// TIA Portal project "T2" (V17)

(* hardware
DEVICE "S7-1500/ET200MP station_1"  S7-1500 station
   slot 0: "Rail_0"  Rack  6ES7 590-1***0-0AA0
   slot 1: "PLC_1"  CPU 1511-1 PN  6ES7 511-1AK01-0AB0  V2.9
      slot 3: "CPU display_1"  6ES7591-1AA00-0AA0
      slot 32768: "PROFINET interface_1"  X1
         slot 32769: "Port_1"  X1 P1
         slot 32770: "Port_2"  X1 P2
      slot 34817: "Virtual CP interface port_1"  Virtual CP interface port  Virtual CP interface port
   slot 2: "DI 32x24VDC SNK/SRC / DQ 32x24VDC/0.3A SNK BA_1"  DI 32x24VDC SNK/SRC / DQ 32x24VDC/0.3A SNK BA  6ES7 523-1BP50-0AA0  V1.0
DEVICE "HMI_1"  TP1500 Comfort PRO
   slot 0: "HMI_1"  TP1500 Comfort PRO  6AV2 124-0QC24-1AXx  17.0.0.0
   slot 1: "HMI_RT_2"  TP1500 Comfort PRO  6AV2 124-0QC24-1AXx  17.0.0.0
   slot 5: "HMI_1.IE_CP_1"  PROFINET Interface  17.0.0.0
      slot 1: "PROFINET Interface_1"  PROFINET Interface
         slot 1: "Port_1"  Port
         slot 2: "Port_2"  Port
   slot 6: "HMI_1.IE_CP_2"  PROFINET Interface  17.0.0.0
      slot 1: "PROFINET Interface_GBit"  PROFINET Interface
         slot 1: "Port_1"  Port
   slot 7: "HMI_1.MPI/DP_CP_1"  MPI/DP Interface  17.0.0.0
*)

// ===== PLC "PLC_1"  CPU 1511-1 PN =====

VAR_GLOBAL   // PLC tag table "Default tag table"
   "System_Byte" AT %MB500 : Byte;
   "FirstScan" AT %M500.0 : Bool;
   "DiagStatusUpdate" AT %M500.1 : Bool;
   "AlwaysTRUE" AT %M500.2 : Bool;
   "AlwaysFALSE" AT %M500.3 : Bool;
   "OPC_Marcha" AT %I0.0 : Bool;
   "OPC_Paro" AT %I0.1 : Bool;
   "Mantenimineto_Fin" AT %M0.0 : Bool;
   "Act_Mantenimiento" AT %M0.1 : Bool;
   "Proceso_Activo" AT %M0.2 : Bool;
   "OPC_SPress_VAC" AT %I0.2 : Bool;
   "OPC_S1_VAC" AT %I0.3 : Bool;
   "OPC_S3_VAC" AT %I0.4 : Bool;
   "OPC_S4_VAC" AT %I0.5 : Bool;
   "OPC_S5_VAC" AT %I0.6 : Bool;
   "OPC_S_VAC_A_Buena" AT %I0.7 : Bool;
   "OPC_S_VAC_A_Mala" AT %I1.0 : Bool;
   "OPC_S_VAC_B" AT %I1.1 : Bool;
   "P_REC_MAQ_CAL_VAC" AT %M0.6 : Bool;
   "P_REC_MAQ_CAL_SOP" AT %M0.7 : Bool;
   "P_REC_MAQ_CAL_EMB" AT %M1.0 : Bool;
   "OPC_Emisor_Vacunas" AT %Q0.0 : Bool;
   "OPC_QC2_VAC" AT %Q0.2 : Bool;
   "OPC_QC3_VAC" AT %Q0.3 : Bool;
   "Pieza_Enviada_MAQ_5_VAC" AT %M3.0 : Bool;
   "VACUNA_ESPERANDO_SOPORTE" AT %M3.2 : Bool;
   "Vacuna_en_Soporte" AT %M3.3 : Bool;
   "Pieza_Enviada_MAQ_5_SOP" AT %M4.1 : Bool;
   "SOPORTE_ESPERANDO_VACUNA" AT %M4.2 : Bool;
   "ACT_EMP_1" AT %M4.6 : Bool;
   "P_Enviada_EMP1" AT %M4.7 : Bool;
   "ACT_EMP_2" AT %M5.0 : Bool;
   "P_Enviada_EMP2" AT %M5.1 : Bool;
   "Transfer_EMP_VACSOP1_Libre" AT %M5.2 : Bool;
   "Transfer_EMP_VACSOP2_Libre" AT %M5.4 : Bool;
   "Vacuna_A" AT %M6.0 : Bool;
   "Vacuna_B" AT %M6.1 : Bool;
   "Soporte_A" AT %M6.2 : Bool;
   "Soporte_B" AT %M6.3 : Bool;
   "Embalaje_A" AT %M6.4 : Bool;
   "Embalaje_B" AT %M6.5 : Bool;
   "Pieza_Enviada_MAQ_5_EMB" AT %M7.2 : Bool;
   "P_Enviada_EMB_EMB" AT %M7.3 : Bool;
   "Cinta_7_EMB_Libre" AT %M7.4 : Bool;
   "Activar_TRansfer_3_EMP" AT %M7.5 : Bool;
   "Act_Cinta_7_EMP" AT %M7.6 : Bool;
   "Transfer_3_EMP_Libre" AT %M7.7 : Bool;
   "Transfer_2_EMP_EMBSOPVAC_Libre" AT %M8.0 : Bool;
   "Trasnfer_2_EMPSOPVAC_Libre" AT %M8.2 : Bool;
   "Trasnfer_1_EMPSOPVAC_Libre" AT %M8.3 : Bool;
   "Act_Maq_1_EMBSOPVAC" AT %M8.4 : Bool;
   "Act_Maq_2_EMBSOPVAC" AT %M8.5 : Bool;
   "EMP1_EMBSOPVAC_Libre" AT %M8.6 : Bool;
   "Esperando_Embalaje" AT %M8.7 : Bool;
   "Vacuna_Lista" AT %M9.4 : Bool;
   "Empaquetar_vacuna" AT %M9.5 : Bool;
   "Empaquetar_Soporte" AT %M9.6 : Bool;
   "Vacuna_Empaquetada" AT %M9.7 : Bool;
   "Soporte_Empaquetado" AT %M10.0 : Bool;
   "Soporte_Listo" AT %M10.1 : Bool;
   "OPC_SETA" AT %I1.2 : Bool;
   "Act_Mantenimiento_Emergencia" AT %M10.2 : Bool;
   "Act_Vaciado" AT %M10.3 : Bool;
   "Emergencia" AT %M10.4 : Bool;
   "Fin_Vaciado" AT %M10.5 : Bool;
   "OPC_Reset" AT %I1.3 : Bool;
   "OPC_Resume" AT %I2.3 : Bool;
   "HMI_Marcha" AT %M10.6 : Bool;
   "ContadorPiezasFinalizadas" AT %MW12 : Int;
   "OPC_QC4_VAC" AT %Q0.4 : Bool;
   "OPC_QC5_VAC" AT %Q0.5 : Bool;
   "OPC_QC6_VAC" AT %Q0.6 : Bool;
   "OPC_QC7_VAC" AT %Q0.7 : Bool;
   "OPC_QTRANS1_VAC" AT %Q1.0 : Bool;
   "OPC_QTRANS2_VAC" AT %Q1.1 : Bool;
   "OPC_QHOR_VAC" AT %Q1.2 : Bool;
   "OPC_QBAJ_VAC" AT %Q1.3 : Bool;
   "OPC_QGRIP_VAC" AT %Q1.4 : Bool;
   "OPC_CLAMP1_VAC" AT %Q1.5 : Bool;
   "HaySoporte" AT %M3.1 : Bool;
   "HayVacuna" AT %M3.4 : Bool;
   "VacunaEnSoporte" AT %M3.5 : Bool;
   "OPC_SPress_SOP" AT %I1.4 : Bool;
   "OPC_S1_SOP" AT %I1.5 : Bool;
   "OPC_S3_SOP" AT %I1.6 : Bool;
   "OPC_S4_SOP" AT %I1.7 : Bool;
   "OPC_S5_SOP" AT %I2.0 : Bool;
   "OPC_S_SOP_A_Buena" AT %I2.1 : Bool;
   "OPC_S_SOP_A_Mala" AT %I2.2 : Bool;
   "OPC_S_SOP_B" AT %I2.4 : Bool;
   "OPC_Emisor_SOP" AT %Q1.7 : Bool;
   "OPC_QC1_SOP" AT %Q2.0 : Bool;
   "OPC_QC2_SOP" AT %Q2.1 : Bool;
   "OPC_QC3_SOP" AT %Q2.2 : Bool;
   "OPC_QC4_SOP" AT %Q2.3 : Bool;
   "OPC_QC5_SOP" AT %Q2.4 : Bool;
   "OPC_QC6_SOP" AT %Q2.5 : Bool;
   "OPC_QC7_SOP" AT %Q2.6 : Bool;
   "OPC_QTRANS1_SOP" AT %Q2.7 : Bool;
   "OPC_QTRANS2_SOP" AT %Q3.0 : Bool;
   "OPC_QHOR_SOP" AT %Q3.1 : Bool;
   "OPC_QBAJ_SOP" AT %Q3.2 : Bool;
   "OPC_QGRIP_SOP" AT %Q3.3 : Bool;
   "OPC_CLAMP1_SOP" AT %Q3.4 : Bool;
   "OPC_SUBCLAMP1_SOP" AT %Q3.5 : Bool;
   "OPC_QC8_SOP" AT %Q3.7 : Bool;
   "OPC_QC9_SOP" AT %Q4.0 : Bool;
   "OPC_QC10_SOP" AT %Q4.1 : Bool;
   "OPC_S6_SOP" AT %I2.5 : Bool;
   "OPC_CLAMP2_SOP" AT %Q4.2 : Bool;
   "OPC_SPress_EMB" AT %I2.6 : Bool;
   "OPC_S1_EMB" AT %I2.7 : Bool;
   "OPC_S3_EMB" AT %I3.0 : Bool;
   "OPC_S4_EMB" AT %I3.1 : Bool;
   "OPC_S5_EMB" AT %I3.2 : Bool;
   "OPC_S_EMB_A_Buena" AT %I3.3 : Bool;
   "OPC_S_EMB_A_Mala" AT %I3.4 : Bool;
   "OPC_S6_EMB" AT %I3.5 : Bool;
   "OPC_Emisor_EMB_Bueno" AT %Q4.3 : Bool;
   "OPC_QC1A_EMB" AT %Q4.4 : Bool;
   "OPC_QC2_EMB" AT %Q4.6 : Bool;
   "OPC_QC3_EMB" AT %Q4.7 : Bool;
   "OPC_QC4_EMB" AT %Q5.0 : Bool;
   "OPC_QC5_EMB" AT %Q5.1 : Bool;
   "OPC_QC6_EMB" AT %Q5.2 : Bool;
   "OPC_QC7_EMB" AT %Q5.3 : Bool;
   "OPC_QTRANS1_EMB" AT %Q5.4 : Bool;
   "OPC_QTRANS2_EMB" AT %Q5.5 : Bool;
   "OPC_S_EMB_B" AT %I3.6 : Bool;
   "OPC_QCLAMP_EMB" AT %Q5.6 : Bool;
   "OPC_QSUBCLAMP_EMB" AT %Q5.7 : Bool;
   "OPC_QTRANS3_EMB" AT %Q6.0 : Bool;
   "OPC_S7_EMB" AT %I3.7 : Bool;
   "Contador_VacunasABuenas" AT %MW14 : Int;
   "Contador_VacunasAMalas" AT %MW16 : Int;
   "Contador_VacunasB" AT %MW18 : Int;
   "Contador_SoportesABuenos" AT %MW26 : Int;
   "Contador_SoportesAMalos" AT %MW28 : Int;
   "Contador_SoportesB" AT %MW36 : Int;
   "Contador_EmbalajesABuenos" AT %MW38 : Int;
   "Contador_EmbalajesAMalos" AT %MW44 : Int;
   "Contador_EmbalajesB" AT %MW46 : Int;
   "MANT_Activar_Cintas" AT %M48.0 : Bool;
   "MANT_Activar_Transfers" AT %M48.1 : Bool;
   "MANT_Activar_Clampers" AT %M48.2 : Bool;
   "MANT_BAJAR_Robots" AT %M48.3 : Bool;
   "MANT_Subir_Clampers" AT %M48.4 : Bool;
   "MANT_Grippers" AT %M48.5 : Bool;
   "MANT_Mover_HOR" AT %M48.6 : Bool;
   "Pieza_Finalizada" AT %M48.7 : Bool;
   "Vac_A_Buena" AT %M49.0 : Bool;
   "VAC_A_Mala" AT %M49.1 : Bool;
   "VAC_B" AT %M49.2 : Bool;
   "SOP_A_Bueno" AT %M49.3 : Bool;
   "SOP_A_Malo" AT %M49.4 : Bool;
   "SOP_B" AT %M49.5 : Bool;
   "EMB_A_Bueno" AT %M49.6 : Bool;
   "EMB_A_Malo" AT %M49.7 : Bool;
   "EMB_B" AT %M50.0 : Bool;
   "Activar_grafcets_vaciados" AT %M50.1 : Bool;
   "fin_vaciado_vac_1" AT %M50.2 : Bool;
   "fin_vaciado_vac_2" AT %M50.3 : Bool;
   "fin_vaciado_vac_3" AT %M50.4 : Bool;
   "fin_vaciado_sop_1" AT %M50.5 : Bool;
   "fin_vaciado_sop_2" AT %M50.6 : Bool;
   "fin_vaciado_sop_3" AT %M50.7 : Bool;
   "fin_vaciado_emb_1" AT %M51.0 : Bool;
   "fin_vaciado_emb_2" AT %M51.1 : Bool;
   "fin_vaciado_emb_3" AT %M51.2 : Bool;
   "fin_vaciado_emb_4" AT %M51.3 : Bool;
   "OPC_SUBCLAMP2_SOP" AT %Q3.6 : Bool;
   "opc_qsubclamp1_vac" AT %Q1.6 : Bool;
   "OPC_Emisor_EMB_Malo" AT %Q6.1 : Bool;
   "Pieza_Rec_maq2emb" AT %M0.3 : Bool;
   "PiezaRecSopMaq2" AT %M25.2 : Bool;
   "PiezaRecVacmaq2" AT %M25.3 : Bool;
   "OPC_QC1_VAC" AT %Q0.1 : Bool;
   "OPC_QC1B_EMB" AT %Q4.5 : Bool;
   "HMI_Resume" AT %M5.3 : Bool;
   "estado_maq1_vac" AT %MW70 : Int;
   "estado_maq2_vac" AT %MW72 : Int;
   "estado_maq3_vac" AT %MW74 : Int;
   "estado_maq4_vac" AT %MW76 : Int;
   "estado_maq5_vac" AT %MW78 : Int;
   "estado_maq1_sop" AT %MW80 : Int;
   "estado_maq2_sop" AT %MW82 : Int;
   "estado_maq3_sop" AT %MW84 : Int;
   "estado_maq4_sop" AT %MW86 : Int;
   "estado_maq5_sop" AT %MW88 : Int;
   "estado_maq6_sop" AT %MW90 : Int;
   "estado_maq1_emb" AT %MW92 : Int;
   "estado_maq2_emb" AT %MW94 : Int;
   "estado_maq3_emb" AT %MW96 : Int;
   "estado_maq4_emb" AT %MW98 : Int;
   "estado_maq5_emb" AT %MW100 : Int;
   "estado_maq6_emb" AT %MW102 : Int;
   "estado_maq7_emb" AT %MW104 : Int;
   "HMI" AT %M6.6 : Bool;
END_VAR

VAR_GLOBAL   // PLC tag table "Manual"
   "Act_Manual_Cinta1_VAC" AT %M30.0 : Bool;
   "Act_Manual_Cinta2_VAC" AT %M30.1 : Bool;
   "Act_Manual_Cinta3_VAC" AT %M30.2 : Bool;
   "Act_Manual_Cinta4_VAC" AT %M30.3 : Bool;
   "Act_Manual_Cinta5_VAC" AT %M30.4 : Bool;
   "Act_Manual_Cinta6_VAC" AT %M30.5 : Bool;
   "Act_Manual_Cinta1_SOP" AT %M30.6 : Bool;
   "Act_Manual_Cinta2_SOP" AT %M30.7 : Bool;
   "Act_Manual_Cinta3_SOP" AT %M31.0 : Bool;
   "Act_Manual_Cinta4_SOP" AT %M31.1 : Bool;
   "Act_Manual_Cinta5_SOP" AT %M31.2 : Bool;
   "Act_Manual_Cinta6_SOP" AT %M31.3 : Bool;
   "Act_Manual_Cinta1_EMB" AT %M31.4 : Bool;
   "Act_Manual_Cinta2_EMB" AT %M31.5 : Bool;
   "Act_Manual_Cinta3_EMB" AT %M31.6 : Bool;
   "Act_Manual_Cinta4_EMB" AT %M31.7 : Bool;
   "Act_Manual_Cinta1_EMP" AT %M32.0 : Bool;
   "Act_Manual_Cinta2_EMP" AT %M32.1 : Bool;
   "Act_Manual_Cinta3_EMP" AT %M32.2 : Bool;
   "Act_Manual_QBAJ1_VAC" AT %M32.3 : Bool;
   "Act_Manual_QBAJ2_VAC" AT %M32.4 : Bool;
   "Act_Manual_QHOR1_VAC" AT %M32.5 : Bool;
   "Act_Manual_QHOR2_VAC" AT %M32.6 : Bool;
   "Act_Manual_QROT1_VAC" AT %M32.7 : Bool;
   "Act_Manual_QGRIP1_VAC" AT %M33.0 : Bool;
   "Act_Manual_QGRIP2_VAC" AT %M33.1 : Bool;
   "Act_Manual_QBAJ1_SOP" AT %M33.2 : Bool;
   "Act_Manual_QBAJ2_SOP" AT %M33.3 : Bool;
   "Act_Manual_QHOR1_SOP" AT %M33.4 : Bool;
   "Act_Manual_QHOR2_SOP" AT %M33.5 : Bool;
   "Act_Manual_QROT1_SOP" AT %M33.6 : Bool;
   "Act_Manual_QGRIP1_SOP" AT %M33.7 : Bool;
   "Act_Manual_QGRIP2_SOP" AT %M34.0 : Bool;
   "Act_Manual_QBAJ1_EMB" AT %M34.1 : Bool;
   "Act_Manual_QHOR1_EMB" AT %M34.2 : Bool;
   "Act_Manual_QGRIP1_EMB" AT %M34.3 : Bool;
END_VAR

VAR_GLOBAL   // PLC tag table "Marcas_Maq_Libre"
   "MAQ1_Libre_VAC" AT %M20.0 : Bool;
   "MAQ2_Libre_VAC" AT %M20.1 : Bool;
   "MAQ3_Libre_VAC" AT %M20.2 : Bool;
   "MAQ4_Libre_VAC" AT %M20.3 : Bool;
   "MAQ5_Libre_VAC" AT %M20.4 : Bool;
   "MAQ1_Libre_SOP" AT %M20.5 : Bool;
   "MAQ2_Libre_SOP" AT %M20.6 : Bool;
   "MAQ3_Libre_SOP" AT %M20.7 : Bool;
   "MAQ4_Libre_SOP" AT %M21.0 : Bool;
   "MAQ5_Libre_SOP" AT %M21.1 : Bool;
   "MAQ1_Libre_EMB" AT %M21.2 : Bool;
   "MAQ2_Libre_EMB" AT %M21.3 : Bool;
   "MAQ3_Libre_EMB" AT %M21.4 : Bool;
   "MAQ4_Libre_EMB" AT %M21.5 : Bool;
   "MAQ5_Libre_EMB" AT %M21.6 : Bool;
   "Act_Maq_2_VAC" AT %M21.7 : Bool;
   "Act_Maq_3_Buena_VAC" AT %M22.0 : Bool;
   "Act_Maq_4_Buena_VAC" AT %M22.1 : Bool;
   "Act_Maq_5_VAC" AT %M22.2 : Bool;
   "Act_Maq_3_Mala_VAC" AT %M22.3 : Bool;
   "Act_Maq_4_Mala_VAC" AT %M22.4 : Bool;
   "Act_Maq_2_SOP" AT %M22.5 : Bool;
   "Act_Maq_3_Buena_SOP" AT %M22.6 : Bool;
   "Act_Maq_4_Buena_SOP" AT %M22.7 : Bool;
   "Act_Maq_5_SOP" AT %M23.0 : Bool;
   "Act_Maq_3_Mala_SOP" AT %M23.1 : Bool;
   "Act_Maq_4_Mala_SOP" AT %M23.2 : Bool;
   "MAQ6_Libre_SOP" AT %M23.3 : Bool;
   "Act_Maq_6_SOP" AT %M23.4 : Bool;
   "HayEmbalaje" AT %M23.5 : Bool;
   "HayVACSOP" AT %M23.6 : Bool;
   "VACSOPEnEMB" AT %M23.7 : Bool;
   "Act_Maq_2_EMB" AT %M24.0 : Bool;
   "Act_Maq_3_Buena_EMB" AT %M24.1 : Bool;
   "Act_Maq_4_Buena_EMB" AT %M24.2 : Bool;
   "Act_Maq_5_EMB" AT %M24.3 : Bool;
   "Act_Maq_3_Mala_EMB" AT %M24.4 : Bool;
   "Act_Maq_4_Mala_EMB" AT %M24.5 : Bool;
   "Act_Maq_6_EMB" AT %M24.6 : Bool;
   "MAQ6_Libre_EMB" AT %M24.7 : Bool;
   "Act_Maq_7_EMB" AT %M25.0 : Bool;
   "MAQ7_Libre_EMB" AT %M25.1 : Bool;
END_VAR

VAR_GLOBAL   // PLC tag table "Marca_Maq_Alarama"
   "Maq1_Alarma_VAC" AT %M40.0 : Bool;
   "Maq2_Alarma_VAC" AT %M40.1 : Bool;
   "Maq3_Alarma_VAC" AT %M40.2 : Bool;
   "Maq4_Alarma_VAC" AT %M40.3 : Bool;
   "Maq5_Alarma_VAC" AT %M40.4 : Bool;
   "Maq1_Alarma_SOP" AT %M40.5 : Bool;
   "Maq2_Alarma_SOP" AT %M40.6 : Bool;
   "Maq3_Alarma_SOP" AT %M40.7 : Bool;
   "Maq4_Alarma_SOP" AT %M41.0 : Bool;
   "Maq5_Alarma_SOP" AT %M41.1 : Bool;
   "Maq6_Alarama_SOP" AT %M41.2 : Bool;
   "Maq1_Alarma_EMB" AT %M41.3 : Bool;
   "Maq2_Alarma_EMB" AT %M41.4 : Bool;
   "Maq3_Alarma_EMB" AT %M41.5 : Bool;
   "Maq4_Alarma_EMB" AT %M41.6 : Bool;
   "Maq5_Alarma_EMB" AT %M41.7 : Bool;
   "Maq6_Alarama_EMB" AT %M42.0 : Bool;
END_VAR

VAR_GLOBAL   // PLC tag table "Marcas_vaciado"
   "vaciado_qc1_vac" AT %M60.0 : Bool;
   "vaciado_qc2_vac" AT %M60.1 : Bool;
   "vaciado_qc3_Vac" AT %M60.2 : Bool;
   "vaciado_qc4_vac" AT %M60.3 : Bool;
   "vaciado_qc5_vac" AT %M60.4 : Bool;
   "vaciado_qc6_vac" AT %M60.5 : Bool;
   "vaciado_qc7_vac" AT %M60.6 : Bool;
   "vaciado_trans1_vac" AT %M60.7 : Bool;
   "vaciado_trans2_vac" AT %M61.0 : Bool;
   "vaciado_subclamp_vac" AT %M61.1 : Bool;
   "vaciado_qc1_sop" AT %M61.2 : Bool;
   "vaciado_qc2_sop" AT %M61.3 : Bool;
   "vaciado_Qc3_sop" AT %M61.4 : Bool;
   "vaciado_Qc4_sop" AT %M61.5 : Bool;
   "vaciado_qc5_sop" AT %M61.6 : Bool;
   "vaciado_Qc6_sop" AT %M61.7 : Bool;
   "vaciado_qc7_sop" AT %M62.0 : Bool;
   "vaciado_Qc8_sop" AT %M62.1 : Bool;
   "vaciado_Qc9_sop" AT %M62.2 : Bool;
   "vaciado_qc10_sop" AT %M62.3 : Bool;
   "vaciado_trasn1_sop" AT %M62.4 : Bool;
   "vaciado_trans2_sop" AT %M62.5 : Bool;
   "vaciado_subclamp1_sop" AT %M62.6 : Bool;
   "vaciado_subclamp2_sop" AT %M62.7 : Bool;
   "vaciado_qc1_emb" AT %M63.0 : Bool;
   "vaciado_Qc2_emb" AT %M63.1 : Bool;
   "vaciado_qc3_emb" AT %M63.2 : Bool;
   "vaciado_Qc4_emb" AT %M63.3 : Bool;
   "vaciado_Qc5_emb" AT %M63.4 : Bool;
   "vaciado_qc6_emb" AT %M63.5 : Bool;
   "vaciado_Qc7_emb" AT %M63.6 : Bool;
   "vaciado_qtrans1_emb" AT %M63.7 : Bool;
   "vaciado_qtrans2_emb" AT %M64.0 : Bool;
   "vaciado_sublcamp2_emb" AT %M64.1 : Bool;
END_VAR

DATA_BLOCK "Grafcet_0_principal_DB"   // DB1
{ S7_Optimized_Access := 'TRUE' }
VERSION : 0.1
// stored: InstanceOfName Grafcet_0_Principal
"Grafcet_0_Principal"
BEGIN
END_DATA_BLOCK

DATA_BLOCK "grafcet_90_EMB"   // DB2
{ S7_Optimized_Access := 'TRUE' }
VERSION : 0.1
// stored: InstanceOfName grafcet_90
"grafcet_90"
BEGIN
END_DATA_BLOCK

DATA_BLOCK "Grafcet_110_Mantenimiento_DB"   // DB3
{ S7_Optimized_Access := 'TRUE' }
VERSION : 0.1
// stored: InstanceOfName Grafcet_110_Mantenimiento
"Grafcet_110_Mantenimiento"
BEGIN
END_DATA_BLOCK

DATA_BLOCK "grafcet_100_EMB"   // DB4
{ S7_Optimized_Access := 'TRUE' }
VERSION : 0.1
// stored: InstanceOfName grafcet_100
"grafcet_100"
BEGIN
END_DATA_BLOCK

DATA_BLOCK "grafcet_120_vaciado_general_DB"   // DB5
{ S7_Optimized_Access := 'TRUE' }
VERSION : 0.1
// stored: InstanceOfName grafcet_120_vaciado_general
"grafcet_120_vaciado_general"
BEGIN
END_DATA_BLOCK

DATA_BLOCK "Grafcet_10_Final_1_EMBV2"   // DB6
{ S7_Optimized_Access := 'TRUE' }
VERSION : 0.1
// stored: InstanceOfName Grafcet_10_Final_1
"Grafcet_10_Final_1"
BEGIN
END_DATA_BLOCK

DATA_BLOCK "grafcet_125_vaciado_tipo1_VAC1"   // DB7
{ S7_Optimized_Access := 'TRUE' }
VERSION : 0.1
// stored: InstanceOfName grafcet_125_vaciado_tipo1
"grafcet_125_vaciado_tipo1"
BEGIN
END_DATA_BLOCK

DATA_BLOCK "grafcet_125_vaciado_tipo1_VAC2"   // DB8
{ S7_Optimized_Access := 'TRUE' }
VERSION : 0.1
// stored: InstanceOfName grafcet_125_vaciado_tipo1
"grafcet_125_vaciado_tipo1"
BEGIN
END_DATA_BLOCK

DATA_BLOCK "grafcet_130_vaciados_maq_VAC3"   // DB9
{ S7_Optimized_Access := 'TRUE' }
VERSION : 0.1
// stored: InstanceOfName grafcet_130_vaciados_maq
"grafcet_130_vaciados_maq"
BEGIN
END_DATA_BLOCK

DATA_BLOCK "grafcet_125_vaciado_tipo1_SOP1"   // DB10
{ S7_Optimized_Access := 'TRUE' }
VERSION : 0.1
// stored: InstanceOfName grafcet_125_vaciado_tipo1
"grafcet_125_vaciado_tipo1"
BEGIN
END_DATA_BLOCK

DATA_BLOCK "grafcet_125_vaciado_tipo1_SOP2"   // DB11
{ S7_Optimized_Access := 'TRUE' }
VERSION : 0.1
// stored: InstanceOfName grafcet_125_vaciado_tipo1
"grafcet_125_vaciado_tipo1"
BEGIN
END_DATA_BLOCK

DATA_BLOCK "grafcet_130_vaciados_maq_SOP3"   // DB12
{ S7_Optimized_Access := 'TRUE' }
VERSION : 0.1
// stored: InstanceOfName grafcet_130_vaciados_maq
"grafcet_130_vaciados_maq"
BEGIN
END_DATA_BLOCK

DATA_BLOCK "grafcet_125_vaciado_tipo1_EMB1"   // DB13
{ S7_Optimized_Access := 'TRUE' }
VERSION : 0.1
// stored: InstanceOfName grafcet_125_vaciado_tipo1
"grafcet_125_vaciado_tipo1"
BEGIN
END_DATA_BLOCK

DATA_BLOCK "grafcet_125_vaciado_tipo1_EMB2"   // DB14
{ S7_Optimized_Access := 'TRUE' }
VERSION : 0.1
// stored: InstanceOfName grafcet_125_vaciado_tipo1
"grafcet_125_vaciado_tipo1"
BEGIN
END_DATA_BLOCK

DATA_BLOCK "grafcet_130_vaciados_maq_EMB3"   // DB15
{ S7_Optimized_Access := 'TRUE' }
VERSION : 0.1
// stored: InstanceOfName grafcet_130_vaciados_maq
"grafcet_130_vaciados_maq"
BEGIN
END_DATA_BLOCK

DATA_BLOCK "grafcet_130_vaciados_maq_EMB4"   // DB16
{ S7_Optimized_Access := 'TRUE' }
VERSION : 0.1
// stored: InstanceOfName grafcet_130_vaciados_maq
"grafcet_130_vaciados_maq"
BEGIN
END_DATA_BLOCK

DATA_BLOCK "Grafcet_1000_Emergencia_"   // DB32
{ S7_Optimized_Access := 'TRUE' }
VERSION : 0.1
// stored: InstanceOfName Grafcet_1000_Emergencia
"Grafcet_1000_Emergencia"
BEGIN
END_DATA_BLOCK

DATA_BLOCK "Grafcet_10_Final_VAC"   // DB52
{ S7_Optimized_Access := 'TRUE' }
VERSION : 0.1
// stored: InstanceOfName Grafcet_10_Final
"Grafcet_10_Final"
BEGIN
END_DATA_BLOCK

DATA_BLOCK "Grafcet_20_FInal_VAC"   // DB53
{ S7_Optimized_Access := 'TRUE' }
VERSION : 0.1
// stored: InstanceOfName Grafcet_20_FInal
"Grafcet_20_FInal"
BEGIN
END_DATA_BLOCK

DATA_BLOCK "grafcet_30_fina_VAC"   // DB54
{ S7_Optimized_Access := 'TRUE' }
VERSION : 0.1
// stored: InstanceOfName grafcet_30_fina
"grafcet_30_fina"
BEGIN
END_DATA_BLOCK

DATA_BLOCK "grafcet_40_final_VAC"   // DB55
{ S7_Optimized_Access := 'TRUE' }
VERSION : 0.1
// stored: InstanceOfName grafcet_40_final
"grafcet_40_final"
BEGIN
END_DATA_BLOCK

DATA_BLOCK "grafcet_50_Final_VAC"   // DB56
{ S7_Optimized_Access := 'TRUE' }
VERSION : 0.1
// stored: InstanceOfName grafcet_50_Final
"grafcet_50_Final"
BEGIN
END_DATA_BLOCK

DATA_BLOCK "Grafcet_70_Final_VAC"   // DB57
{ S7_Optimized_Access := 'TRUE' }
VERSION : 0.1
// stored: InstanceOfName Grafcet_70_Final
"Grafcet_70_Final"
BEGIN
END_DATA_BLOCK

DATA_BLOCK "Grafcet_20_FInal_SOP"   // DB58
{ S7_Optimized_Access := 'TRUE' }
VERSION : 0.1
// stored: InstanceOfName Grafcet_20_FInal
"Grafcet_20_FInal"
BEGIN
END_DATA_BLOCK

DATA_BLOCK "Grafcet_10_Final_SOP"   // DB59
{ S7_Optimized_Access := 'TRUE' }
VERSION : 0.1
// stored: InstanceOfName Grafcet_10_Final
"Grafcet_10_Final"
BEGIN
END_DATA_BLOCK

DATA_BLOCK "grafcet_30_fina_SOP"   // DB60
{ S7_Optimized_Access := 'TRUE' }
VERSION : 0.1
// stored: InstanceOfName grafcet_30_fina
"grafcet_30_fina"
BEGIN
END_DATA_BLOCK

DATA_BLOCK "grafcet_40_final_SOP"   // DB61
{ S7_Optimized_Access := 'TRUE' }
VERSION : 0.1
// stored: InstanceOfName grafcet_40_final
"grafcet_40_final"
BEGIN
END_DATA_BLOCK

DATA_BLOCK "Grafcet_70_Final_SOP"   // DB62
{ S7_Optimized_Access := 'TRUE' }
VERSION : 0.1
// stored: InstanceOfName Grafcet_70_Final
"Grafcet_70_Final"
BEGIN
END_DATA_BLOCK

DATA_BLOCK "grafcet_50_Final_SOP"   // DB63
{ S7_Optimized_Access := 'TRUE' }
VERSION : 0.1
// stored: InstanceOfName grafcet_50_Final
"grafcet_50_Final"
BEGIN
END_DATA_BLOCK

DATA_BLOCK "Grafcet_10_Final_EMB"   // DB64
{ S7_Optimized_Access := 'TRUE' }
VERSION : 0.1
// stored: InstanceOfName Grafcet_10_Final
"Grafcet_10_Final"
BEGIN
END_DATA_BLOCK

DATA_BLOCK "Grafcet_20_2_FInal_EMB"   // DB65
{ S7_Optimized_Access := 'TRUE' }
VERSION : 0.1
// stored: InstanceOfName Grafcet_20_2_FInal
"Grafcet_20_2_FInal"
BEGIN
END_DATA_BLOCK

DATA_BLOCK "grafcet_30_fina_EMB"   // DB66
{ S7_Optimized_Access := 'TRUE' }
VERSION : 0.1
// stored: InstanceOfName grafcet_30_fina
"grafcet_30_fina"
BEGIN
END_DATA_BLOCK

DATA_BLOCK "grafcet_40_final_EMB"   // DB67
{ S7_Optimized_Access := 'TRUE' }
VERSION : 0.1
// stored: InstanceOfName grafcet_40_final
"grafcet_40_final"
BEGIN
END_DATA_BLOCK

DATA_BLOCK "grafcte_80_final_EMB"   // DB68
{ S7_Optimized_Access := 'TRUE' }
VERSION : 0.1
// stored: InstanceOfName grafcte_80_final
"grafcte_80_final"
BEGIN
END_DATA_BLOCK

DATA_BLOCK "Grafcet_70_Final_EMB"   // DB69
{ S7_Optimized_Access := 'TRUE' }
VERSION : 0.1
// stored: InstanceOfName Grafcet_70_Final
"Grafcet_70_Final"
BEGIN
END_DATA_BLOCK

FUNCTION_BLOCK "Grafcet_0_Principal"   // FB1, SCL
{ S7_Optimized_Access := 'TRUE' }
VERSION : 0.1
   VAR_INPUT
      Paro : Bool;
      HMI_Paro : Bool;
      Marcha : Bool;
      HMI_Marcha : Bool;
      Mantenimiento_Fin : Bool;
      Modo_Manual : Bool;
      Pieza_Empaquetada : Bool;
      CI : Bool;
      VacunaABuena : Bool;
      VacunaAMala : Bool;
      VacunaB : Bool;
      SoporteABueno : Bool;
      SoporteAMalo : Bool;
      SoporteB : Bool;
      EmbalajeABuneo : Bool;
      EmbalajeAMalo : Bool;
      EmbalajeB : Bool;
   END_VAR
   VAR_OUTPUT
      Act_Mantenimiento : Bool;
      Proceso_Activo : Bool;
      Modo_Manual_Activado : Bool;
      contador : Int;
      C_VACAB : Int;
      C_VACAM : Int;
      C_VACB : Int;
      C_SOPAB : Int;
      C_SOPAM : Int;
      C_SOPB : Int;
      C_EMBAB : Int;
      C_EMBAM : Int;
      C_EMBB : Int;
   END_VAR
   VAR
      S0 : Bool;
      S1 : Bool;
      S2 : Bool;
      X0 : Bool;
      X1 : Bool;
      X2 : Bool;
      X3 : Bool;
      S4 : Bool;
      X4 : Bool;
      STOP_NEG : Bool;
      S3 : Bool;
      Paro_Ciclo : Bool;
      S0p : Bool;
      S10e : Bool;
      S11e : Bool;
      S12e : Bool;
      X10e : Bool;
      S1p : Bool;
      X11e : Bool;
      X0p : Bool;
      FORCE_CURRENT_E : Bool;
      FORCE_INIT_E : Bool;
      X12e : Bool;
      X1p : Bool;
      TrigX3 : R_TRIG;
      TrigVACAB : R_TRIG;
      TrigVACAM : R_TRIG;
      TrigVACB : R_TRIG;
      TrigSOPAB : R_TRIG;
      TrigSOPAM : R_TRIG;
      TrigSOPB : R_TRIG;
      TrigEMBAB : R_TRIG;
      TrigEMBAM : R_TRIG;
      TrigEMBB : R_TRIG;
   END_VAR
   VAR RETAIN
      Contador_G : CTU_INT;
      Contador_VACAB : CTU_INT;
      Contador_VACAM : CTU_INT;
      Contador_VACB : CTU_INT;
      Contador_SOPAB : CTU_INT;
      Contador_SOPAM : CTU_INT;
      Contador_SOPB : CTU_INT;
      Contador_EMBAB : CTU_INT;
      Contador_EMBAM : CTU_INT;
      Contador_EMBB : CTU_INT;
   END_VAR
BEGIN

   // EMERGENCIA
   #S10e := (#X12e AND #CI) OR "FirstScan";
   #S11e := #X10e AND "Emergencia";
   #S12e := #X11e;

   #X10e := #S10e OR (#X10e AND NOT #S11e);
   #X11e := #S11e OR (#X11e AND NOT #S12e);
   #X12e := #S12e OR (#X12e AND NOT #S10e);

   #FORCE_INIT_E := #X11e;
   #FORCE_CURRENT_E := #X12e;

   #STOP_NEG := NOT #Paro;

   #S0p := ("FirstScan" OR #X0) AND NOT #FORCE_CURRENT_E;
   #S1p := #X0 AND (#STOP_NEG OR #HMI_Paro) AND NOT #FORCE_CURRENT_E;

   #X0p := (#S0p OR #X0p AND NOT #S1p) AND NOT #FORCE_INIT_E;
   #X1p := (#S1p OR #X1p AND NOT #S0p) AND NOT #FORCE_INIT_E;


   #Paro_Ciclo := #X1p;

   //Grafcet principal
   #S0 := ("FirstScan" OR (#X3 AND #Paro_Ciclo) OR (#X4 AND NOT #Modo_Manual)) AND NOT #FORCE_CURRENT_E;
   #S1 := #X0 AND ((#Marcha OR #HMI_Marcha)AND NOT #Modo_Manual) AND NOT #FORCE_CURRENT_E;
   #S2 := (#X1 AND #Mantenimiento_Fin) OR (#X3 AND NOT #Paro_Ciclo) AND NOT #FORCE_CURRENT_E;
   #S3 := (#X2 AND #Pieza_Empaquetada) AND NOT #FORCE_CURRENT_E;
   #S4 := (#X0 AND #Modo_Manual) AND NOT #FORCE_CURRENT_E;

   #X0 := (#S0 OR #X0 AND (NOT #S1 AND NOT #S4)) OR #FORCE_INIT_E;
   #X1 := (#S1 OR #X1 AND (NOT #S2)) AND NOT #FORCE_INIT_E;
   #X2 := (#S2 OR #X2 AND (NOT #S3)) AND NOT #FORCE_INIT_E;
   #X3 := (#S3 OR #X3 AND (NOT #S0)) AND NOT #FORCE_INIT_E;
   #X4 := (#S4 OR #X4 AND (NOT #S0)) AND NOT #FORCE_INIT_E;

   #Act_Mantenimiento := #X1;
   #Proceso_Activo := #X2 OR #X3;
   #Modo_Manual_Activado := #X4;



   #TrigX3(CLK:=#X3);
   #TrigVACAB(CLK := (#X3 OR #X2) AND #VacunaABuena);
   #TrigVACAM(CLK := (#X3 OR #X2) AND #VacunaAMala);
   #TrigVACB(CLK := (#X3 OR #X2) AND #VacunaB);
   #TrigSOPAB(CLK := (#X3 OR #X2) AND #SoporteABueno);
   #TrigSOPAM(CLK := (#X3 OR #X2) AND #SoporteAMalo);
   #TrigSOPB(CLK := (#X3 OR #X2) AND #SoporteB);
   #TrigEMBAB(CLK := (#X3 OR #X2) AND #EmbalajeABuneo);
   #TrigEMBAM(CLK := (#X3 OR #X2) AND #EmbalajeAMalo);
   #TrigEMBB(CLK := (#X3 OR #X2) AND #EmbalajeB);

   #Contador_G(CU:=#TrigX3.Q,
               R:=#X0,
               PV:=50,
               CV=>#contador);

   #Contador_VACAB(CU := #TrigVACAB.Q,
               R := #X0,
               PV := 50,
               CV => #C_VACAB);

   #Contador_VACAM(CU := #TrigVACAM.Q,
               R := #X0,
               PV := 50,
               CV => #C_VACAM);

   #Contador_VACB(CU := #TrigVACB.Q,
                   R := #X0,
                   PV := 50,
                   CV => #C_VACB);

    #Contador_SOPAB(CU := #TrigSOPAB.Q,
                   R := #X0,
                   PV := 50,
                   CV => #C_SOPAB);

   #Contador_SOPAM(CU := #TrigSOPAM.Q,
                   R := #X0,
                   PV := 50,
                   CV => #C_SOPAM);

   #Contador_SOPB(CU := #TrigSOPB.Q,
                   R := #X0,
                   PV := 50,
                   CV => #C_SOPB);

    #Contador_EMBAB(CU := #TrigEMBAB.Q,
                   R := #X0,
                   PV := 50,
                   CV => #C_EMBAB);

   #Contador_EMBAM(CU := #TrigEMBAM.Q,
                   R := #X0,
                   PV := 50,
                   CV => #C_EMBAM);
   #Contador_EMBB(CU := #TrigEMBB.Q,
                   R := #X0,
                   PV := 50,
                   CV => #C_EMBB);
END_FUNCTION_BLOCK

FUNCTION_BLOCK "grafcte_80_final"   // FB2, SCL
{ S7_Optimized_Access := 'TRUE' }
VERSION : 0.1
   VAR_INPUT
      Act_Proceso : Bool;
      S5 : Bool;
      SigMaqLibre : Bool;
      Mantenimiento_Cinta : Bool;
      vaciado_cinta : Bool;
      CI : Bool;
      Reset : Bool;
      Resume : Bool;
   END_VAR
   VAR_OUTPUT
      Maq_Libre : Bool;
      QC3 : Bool;
      Act_Sig_Maq : Bool;
      Alarma_Maquina : Bool;
   END_VAR
   VAR_IN_OUT
      Alarma_1 : Bool;
      Alarma_2 : Bool;
   END_VAR
   VAR
      S80 : Bool;
      S81 : Bool;
      S82 : Bool;
      S83 : Bool;
      X80 : Bool;
      X81 : Bool;
      X82 : Bool;
      X83 : Bool;
      S80e : Bool;
      S81e : Bool;
      S82e : Bool;
      X80e : Bool;
      X81e : Bool;
      X82e : Bool;
      S80a : Bool;
      S81a : Bool;
      S82a : Bool;
      S83a : Bool;
      X80a : Bool;
      X81a : Bool;
      X82a : Bool;
      X83a : Bool;
      FORCE_INIT : Bool;
      FORCE_INIT_E : Bool;
      FORCE_CURRENT_E : Bool;
      FORCE_CURRENT : Bool;
      STOP_ACT : Bool;
      RESET_ALARMA : Bool;
      Alarma : Bool;
      T1a : TON_TIME;
      T2a : TON_TIME;
   END_VAR
BEGIN
   //Flancos


   // EMERGENCIA
   #S80e := (#X82e AND #CI) OR "FirstScan";
   #S81e := #X80e AND "Emergencia";
   #S82e := #X81e;

   #X80e := #S80e OR (#X80e AND NOT #S81e);
   #X81e := #S81e OR (#X81e AND NOT #S82e);
   #X82e := #S82e OR (#X82e AND NOT #S80e);

   #FORCE_INIT_E := #X81e;
   #FORCE_CURRENT_E := #X82e;


   // ALARMAS
   #S80a := (#X83a AND NOT #FORCE_CURRENT_E) OR "FirstScan";
   #S81a := (#X80a AND #Alarma) AND NOT #FORCE_CURRENT_E;
   #S82a := (#X81a AND #Reset) AND NOT #FORCE_CURRENT_E;
   #S83a := (#X82a OR (#X81a AND #Resume)) AND NOT #FORCE_CURRENT_E;

   #X80a := #S80a OR (#X80a AND NOT #S81a) OR #FORCE_INIT_E;
   #X81a := (#S81a OR (#X81a AND NOT #S82a AND NOT #S83a)) AND NOT #FORCE_INIT_E;
   #X82a := (#S82a OR (#X82a AND NOT #S83a)) AND NOT #FORCE_INIT_E;
   #X83a := (#S83a OR (#X83a AND NOT #S80a)) AND NOT #FORCE_INIT_E;

   #STOP_ACT := #X81a;
   #FORCE_INIT := #FORCE_INIT_E OR #X82a;
   #FORCE_CURRENT := #FORCE_CURRENT_E OR #X81a;
   #RESET_ALARMA := #X83a;




   // PRODUCCIÓN
   #S80 := ("FirstScan" OR (#X83 AND NOT #S5)) AND NOT #FORCE_CURRENT;
   #S81 := (#X80 AND #Act_Proceso) AND NOT #FORCE_CURRENT;
   #S82 := (#X81 AND #S5) AND NOT #FORCE_CURRENT;
   #S83 := (#X82 AND #SigMaqLibre) AND NOT #FORCE_CURRENT;



   #X80 := (#S80 OR #X80 AND (NOT #S81)) OR #FORCE_INIT;
   #X81 := (#S81 OR #X81 AND (NOT #S82)) AND NOT #FORCE_INIT;
   #X82 := (#S82 OR #X82 AND (NOT #S83)) AND NOT #FORCE_INIT;
   #X83 := (#S83 OR #X83 AND (NOT #S80)) AND NOT #FORCE_INIT;



   #Maq_Libre := #X80 AND NOT #STOP_ACT;
   #QC3 := (#X81 OR #X83 OR #Mantenimiento_Cinta OR #vaciado_cinta) AND NOT #STOP_ACT;
   #Act_Sig_Maq := #X83 AND NOT #STOP_ACT;

   #T1a(IN:=#X81,
        PT:=T#5s);
   #T2a(IN := #X83,
        PT := T#5s);


   //#Alarma_1 := (#Alarma_1 OR #T1a.Q) AND NOT #RESET_ALARMA;
   //#Alarma_2 := (#Alarma_2 OR #T2a.Q) AND NOT #RESET_ALARMA;

   //#Alarma := (#Alarma_1 OR #Alarma_2 ) AND NOT (#FORCE_INIT OR #RESET_ALARMA);
END_FUNCTION_BLOCK

FUNCTION_BLOCK "grafcet_90"   // FB3, SCL
{ S7_Optimized_Access := 'TRUE' }
VERSION : 0.1
   VAR_INPUT
      Act_Proceso : Bool;
      SENSOR : Bool;
      SigMaqLibre : Bool;
      Mantenimiento_Cinta : Bool;
      Mantenimiento_Trans : Bool;
      vaicado_cinta : Bool;
      vaciado_trnas : Bool;
      CI : Bool;
      Reset : Bool;
      Resume : Bool;
   END_VAR
   VAR_OUTPUT
      Maq_Libre : Bool;
      QC3 : Bool;
      QTrans : Bool;
      Act_Sig_Maq : Bool;
      Alarma_Maquina : Bool;
   END_VAR
   VAR_IN_OUT
      Alarma_1 : Bool;
      Alarma_2 : Bool;
   END_VAR
   VAR
      S90 : Bool;
      S91 : Bool;
      S92 : Bool;
      S93 : Bool;
      S94 : Bool;
      X90 : Bool;
      X91 : Bool;
      X92 : Bool;
      X93 : Bool;
      X94 : Bool;
      S90e : Bool;
      S91e : Bool;
      S92e : Bool;
      X90e : Bool;
      X91e : Bool;
      X92e : Bool;
      S90a : Bool;
      S91a : Bool;
      S92a : Bool;
      S93a : Bool;
      X90a : Bool;
      X91a : Bool;
      X92a : Bool;
      X93a : Bool;
      Alarma : Bool;
      FORCE_INIT : Bool;
      FORCE_INIT_E : Bool;
      FORCE_CURRENT : Bool;
      FORCE_CURRENT_E : Bool;
      STOP_ACT : Bool;
      RESET_ALARMA : Bool;
      T1a : TON_TIME;
      T2a : TON_TIME;
   END_VAR
BEGIN
   //Flancos


   // EMERGENCIA
   #S90e := (#X92e AND #CI) OR "FirstScan";
   #S91e := #X90e AND "Emergencia";
   #S92e := #X91e;

   #X90e := #S90e OR (#X90e AND NOT #S91e);
   #X91e := #S91e OR (#X91e AND NOT #S92e);
   #X92e := #S92e OR (#X92e AND NOT #S90e);

   #FORCE_INIT_E := #X91e;
   #FORCE_CURRENT_E := #X92e;


   // ALARMAS
   #S90a := (#X93a AND NOT #FORCE_CURRENT_E) OR "FirstScan";
   #S91a := (#X90a AND #Alarma) AND NOT #FORCE_CURRENT_E;
   #S92a := (#X91a AND #Reset) AND NOT #FORCE_CURRENT_E;
   #S93a := (#X92a OR (#X91a AND #Resume)) AND NOT #FORCE_CURRENT_E;

   #X90a := #S90a OR (#X90a AND NOT #S91a) OR #FORCE_INIT_E;
   #X91a := (#S91a OR (#X91a AND NOT #S92a AND NOT #S93a)) AND NOT #FORCE_INIT_E;
   #X92a := (#S92a OR (#X92a AND NOT #S93a)) AND NOT #FORCE_INIT_E;
   #X93a := (#S93a OR (#X93a AND NOT #S90a)) AND NOT #FORCE_INIT_E;

   #STOP_ACT := #X91a;
   #FORCE_INIT := #FORCE_INIT_E OR #X92a;
   #FORCE_CURRENT := #FORCE_CURRENT_E OR #X91a;
   #RESET_ALARMA := #X93a;




   // PRODUCCIÓN
   #S90 := ("FirstScan" OR (#X94)) AND NOT #FORCE_CURRENT;
   #S91 := (#X90 AND #Act_Proceso) AND NOT #FORCE_CURRENT;
   #S92 := (#X91 AND #SENSOR) AND NOT #FORCE_CURRENT;
   #S93 := (#X92 AND #SigMaqLibre) AND NOT #FORCE_CURRENT;
   #S94 := (#X93 AND NOT #SENSOR) AND NOT #FORCE_CURRENT;



   #X90 := (#S90 OR #X90 AND (NOT #S91)) OR #FORCE_INIT;
   #X91 := (#S91 OR #X91 AND (NOT #S92)) AND NOT #FORCE_INIT;
   #X92 := (#S92 OR #X92 AND (NOT #S93)) AND NOT #FORCE_INIT;
   #X93 := (#S93 OR #X93 AND (NOT #S94)) AND NOT #FORCE_INIT;
   #X94 := (#S94 OR #X94 AND (NOT #S90)) AND NOT #FORCE_INIT;



   #Maq_Libre := #X90 AND NOT #STOP_ACT;
   #QC3 := (#X91 OR #Mantenimiento_Cinta OR #vaicado_cinta) AND NOT #STOP_ACT;
   #QTrans := (#X93 OR #Mantenimiento_Trans OR #vaciado_trnas) AND NOT #STOP_ACT;
   #Act_Sig_Maq := #X94 AND NOT #STOP_ACT;

   #T1a(IN:=#X91,
        PT:=T#5s);
   #T2a(IN := #X93,
        PT := T#5s);



   //#Alarma_1 := (#Alarma_1 OR #T1a.Q) AND NOT #RESET_ALARMA;
   //#Alarma_2 := (#Alarma_2 OR #T2a.Q) AND NOT #RESET_ALARMA;

   //#Alarma := (#Alarma_1 OR #Alarma_2) AND NOT (#FORCE_INIT OR #RESET_ALARMA);
END_FUNCTION_BLOCK

FUNCTION_BLOCK "grafcet_100"   // FB4, SCL
{ S7_Optimized_Access := 'TRUE' }
VERSION : 0.1
   VAR_INPUT
      Act_Proceso : Bool;
      S5 : Bool;
      Pieza_Empaquetada : Bool;
      Mantenimiento_Cinta : Bool;
      Mantenimiento_Clamper : Bool;
      Mantenimiento_SubirClamp : Bool;
      vaciado_cinta : Bool;
      vaciado_subclamp : Bool;
      CI : Bool;
      Reset : Bool;
      Resume : Bool;
   END_VAR
   VAR_OUTPUT
      Maq_Libre : Bool;
      QC7 : Bool;
      QCLAMP : Bool;
      QCLAMP_SUB : Bool;
      HayPieza : Bool;
      Pieza_Entregada : Bool;
      Alarma_Maquina : Bool;
   END_VAR
   VAR_IN_OUT
      Alarma_1 : Bool;
   END_VAR
   VAR
      S100 : Bool;
      S101 : Bool;
      S102 : Bool;
      S103 : Bool;
      S104 : Bool;
      S105 : Bool;
      S106 : Bool;
      X100 : Bool;
      X102 : Bool;
      X101 : Bool;
      X103 : Bool;
      X104 : Bool;
      X105 : Bool;
      X106 : Bool;
      S100e : Bool;
      S101e : Bool;
      S102e : Bool;
      X100e : Bool;
      X101e : Bool;
      X102e : Bool;
      S100a : Bool;
      S101a : Bool;
      S102a : Bool;
      S103a : Bool;
      X100a : Bool;
      X101a : Bool;
      X102a : Bool;
      X103a : Bool;
      FORCE_CURRENT_E : Bool;
      FORCE_CURRENT : Bool;
      FORCE_INIT : Bool;
      FORCE_INIT_E : Bool;
      STOP_ACT : Bool;
      RESET_ALARMA : Bool;
      Alarma : Bool;
      S107 : Bool;
      X107 : Bool;
      T1 : TON_TIME;
      T2 : TON_TIME;
      T3 : TON_TIME;
      Trig105 : R_TRIG;
   END_VAR
   VAR RETAIN
      "Counter" : CTU_INT;
   END_VAR
   VAR
      T1a : TON_TIME;
   END_VAR
BEGIN
   //Flancos


   // EMERGENCIA
   #S100e := (#X102e AND #CI) OR "FirstScan";
   #S101e := #X100e AND "Emergencia";
   #S102e := #X101e;

   #X100e := #S100e OR (#X100e AND NOT #S101e);
   #X101e := #S101e OR (#X101e AND NOT #S102e);
   #X102e := #S102e OR (#X102e AND NOT #S100e);

   #FORCE_INIT_E := #X101e;
   #FORCE_CURRENT_E := #X102e;


   // ALARMAS
   #S100a := (#X103a AND NOT #FORCE_CURRENT_E) OR "FirstScan";
   #S101a := (#X100a AND #Alarma) AND NOT #FORCE_CURRENT_E;
   #S102a := (#X101a AND #Reset) AND NOT #FORCE_CURRENT_E;
   #S103a := (#X102a OR (#X101a AND #Resume)) AND NOT #FORCE_CURRENT_E;

   #X100a := #S100a OR (#X100a AND NOT #S101a) OR #FORCE_INIT_E;
   #X101a := (#S101a OR (#X101a AND NOT #S102a AND NOT #S103a)) AND NOT #FORCE_INIT_E;
   #X102a := (#S102a OR (#X102a AND NOT #S103a)) AND NOT #FORCE_INIT_E;
   #X103a := (#S103a OR (#X103a AND NOT #S100a)) AND NOT #FORCE_INIT_E;

   #STOP_ACT := #X101a;
   #FORCE_INIT := #FORCE_INIT_E OR #X102a;
   #FORCE_CURRENT := #FORCE_CURRENT_E OR #X101a;
   #RESET_ALARMA := #X103a;
   #T1(IN:=#X102,
       PT:=T#1s
   );
   #T2(IN := #X103,
       PT := T#1s
   );
   #T3(IN := #X106,
       PT := T#3s
   );

   #Trig105(CLK:=#X105);


   #Counter(CU:=#Trig105.Q,
            R:= #X100,
            PV:=2);



   // PRODUCCIÓN
   #S100 := ("FirstScan" OR (#X107)) AND NOT #FORCE_CURRENT;
   #S101 := (#X100 AND #Act_Proceso) AND NOT #FORCE_CURRENT;
   #S102 := (#X101 AND #S5) AND NOT #FORCE_CURRENT;
   #S103 := (#X102 AND #T1.Q) AND NOT #FORCE_CURRENT;
   #S104 := (#X103 AND #T2.Q) OR (#X105 AND #Counter.CV < 2) AND NOT #FORCE_CURRENT;
   #S105 := (#X104 AND #Pieza_Empaquetada) AND NOT #FORCE_CURRENT;
   #S106 := (#X105 AND #Counter.CV = 2) AND NOT #FORCE_CURRENT;
   #S107 := (#X106 AND #T3.Q) AND NOT #FORCE_CURRENT;


   #X100 := (#S100 OR #X100 AND (NOT #S101)) OR #FORCE_INIT;
   #X101 := (#S101 OR #X101 AND (NOT #S102)) AND NOT #FORCE_INIT;
   #X102 := (#S102 OR #X102 AND (NOT #S103)) AND NOT #FORCE_INIT;
   #X103 := (#S103 OR #X103 AND (NOT #S104)) AND NOT #FORCE_INIT;
   #X104 := (#S104 OR #X104 AND (NOT #S105)) AND NOT #FORCE_INIT;
   #X105 := (#S105 OR #X105 AND (NOT #S106 AND NOT #S104)) AND NOT #FORCE_INIT;
   #X106 := (#S106 OR #X106 AND (NOT #S107)) AND NOT #FORCE_INIT;
   #X107 := (#S107 OR #X107 AND (NOT #S100)) AND NOT #FORCE_INIT;


   #Maq_Libre := #X100 AND NOT #STOP_ACT;

   #QC7 := (#X101 OR #X102 OR #X106 OR #Mantenimiento_Cinta OR #vaciado_cinta) AND NOT #STOP_ACT;
   #QCLAMP := (#X103 OR #Mantenimiento_Clamper ) AND NOT #STOP_ACT;
   #QCLAMP_SUB := (#X106 OR #Mantenimiento_SubirClamp OR #vaciado_subclamp) AND NOT #STOP_ACT;
   #HayPieza := #X104 AND NOT #STOP_ACT;
   #Pieza_Entregada := #X107;

   #T1a(IN := #X101,
        PT := T#15s);


   //#Alarma_1 := (#Alarma_1 OR (#X101 AND #T1a.Q)) AND NOT #RESET_ALARMA;

   //#Alarma := (#Alarma_1 ) AND NOT (#FORCE_INIT OR #RESET_ALARMA);
   //#Alarma_Maquina := #Alarma;
END_FUNCTION_BLOCK

FUNCTION_BLOCK "Grafcet_110_Mantenimiento"   // FB5, SCL
{ S7_Optimized_Access := 'TRUE' }
VERSION : 0.1
   VAR_INPUT
      Act_Mantenimiento : Bool;
      Act_Mantenimiento_Emergencia : Bool;
      CI : Bool;
      Reset : Bool;
      Resume : Bool;
   END_VAR
   VAR_OUTPUT
      Mantenimiento_Activado : Bool;
      Activar_Cintas : Bool;
      Activar_Transfers : Bool;
      BAJAR_ROBOTS : Bool;
      SUBIR_CLAMPERS : Bool;
      GRIPPERS : Bool;
      CLAMPER : Bool;
      MOVER_HOR : Bool;
      Fin_Mantenimiento : Bool;
   END_VAR
   VAR
      X110 : Bool;
      X111 : Bool;
      X112 : Bool;
      X113 : Bool;
      X114 : Bool;
      X115 : Bool;
      X116 : Bool;
      X117 : Bool;
      S110 : Bool;
      S111 : Bool;
      S112 : Bool;
      S113 : Bool;
      S114 : Bool;
      S115 : Bool;
      S116 : Bool;
      S117 : Bool;
      Sensores : Bool;
      FORCE_CURRENT : Bool;
      FORCE_CURRENT_E : Bool;
      FORCE_INIT : Bool;
      FORCE_INIT_E : Bool;
      STOP_ACT : Bool;
      S110e : Bool;
      S111e : Bool;
      S112e : Bool;
      X110e : Bool;
      X111e : Bool;
      X112e : Bool;
      S110a : Bool;
      S111a : Bool;
      S112a : Bool;
      S113a : Bool;
      X110a : Bool;
      X111a : Bool;
      X112a : Bool;
      X113a : Bool;
      Alarma : Bool;
      RESET_ALARMA : Bool;
      T1 : TON_TIME;
      T2 : TON_TIME;
      T3 : TON_TIME;
      T4 : TON_TIME;
      T5 : TON_TIME;
   END_VAR
BEGIN
   //Flancos


   // EMERGENCIA
   #S110e := (#X112e AND #CI) OR "FirstScan";
   #S111e := #X110e AND FALSE;
   #S112e := #X111e;

   #X110e := #S110e OR (#X110e AND NOT #S111e);
   #X111e := #S111e OR (#X111e AND NOT #S112e);
   #X112e := #S112e OR (#X112e AND NOT #S110e);

   #FORCE_INIT_E := #X111e;
   #FORCE_CURRENT_E := #X112e;


   // ALARMAS
   #S110a := (#X113a AND NOT #FORCE_CURRENT_E) OR "FirstScan";
   #S111a := (#X110a AND #Alarma) AND NOT #FORCE_CURRENT_E;
   #S112a := (#X111a AND #Reset) AND NOT #FORCE_CURRENT_E;
   #S113a := (#X112a OR (#X111a AND #Resume)) AND NOT #FORCE_CURRENT_E;

   #X110a := #S110a OR (#X110a AND NOT #S111a) OR #FORCE_INIT_E;
   #X111a := (#S111a OR (#X111a AND NOT #S112a AND NOT #S113a)) AND NOT #FORCE_INIT_E;
   #X112a := (#S112a OR (#X112a AND NOT #S113a)) AND NOT #FORCE_INIT_E;
   #X113a := (#S113a OR (#X113a AND NOT #S110a)) AND NOT #FORCE_INIT_E;

   #STOP_ACT := #X111a;
   #FORCE_INIT := #FORCE_INIT_E OR #X112a;
   #FORCE_CURRENT := #FORCE_CURRENT_E OR #X111a;
   #RESET_ALARMA := #X113a;


   #T1(IN:=#X112,
       PT:=T#2s
   );
   #T2(IN := #X113,
       PT := T#2s
   );
   #T3(IN := #X114,
       PT := T#2s
   );
   #T4(IN := #X115,
       PT := T#2s
   );
   #T5(IN := #X116,
       PT := T#2s
   );


   #Sensores := FALSE;

   // PRODUCCIÓN
   #S110 := ("FirstScan" OR (#X117)) AND NOT #FORCE_CURRENT;
   //#S111 := (#X110 AND (#Act_Mantenimiento OR #Act_Mantenimiento_Emergencia)) AND NOT #FORCE_CURRENT;
   #S111 := (#X110 AND (#Act_Mantenimiento OR #Act_Mantenimiento_Emergencia) ) AND NOT #FORCE_CURRENT;
   #S112 := (#X111 AND NOT #Sensores) AND NOT #FORCE_CURRENT;
   #S113 := (#X112 AND #T1.Q) AND NOT #FORCE_CURRENT;
   #S114 := (#X113 AND #T2.Q) AND NOT #FORCE_CURRENT;
   #S115 := (#X114 AND #T3.Q) AND NOT #FORCE_CURRENT;
   #S116 := (#X115 AND #T4.Q) AND NOT #FORCE_CURRENT;
   #S117 := (#X116 AND #T5.Q) AND NOT #FORCE_CURRENT;


   #X110 := (#S110 OR #X110 AND (NOT #S111)) OR #FORCE_INIT;
   #X111 := (#S111 OR #X111 AND (NOT #S112)) AND NOT #FORCE_INIT;
   #X112 := (#S112 OR #X112 AND (NOT #S113)) AND NOT #FORCE_INIT;
   #X113 := (#S113 OR #X113 AND (NOT #S114)) AND NOT #FORCE_INIT;
   #X114 := (#S114 OR #X114 AND (NOT #S115)) AND NOT #FORCE_INIT;
   #X115 := (#S115 OR #X115 AND (NOT #S116)) AND NOT #FORCE_INIT;
   #X116 := (#S116 OR #X116 AND (NOT #S117)) AND NOT #FORCE_INIT;
   #X117 := (#S117 OR #X117 AND (NOT #S110)) AND NOT #FORCE_INIT;

   #Activar_Cintas := #X112 AND NOT #STOP_ACT;
   #Activar_Transfers := #X113 AND NOT #STOP_ACT;
   #BAJAR_ROBOTS := #X114 AND NOT #STOP_ACT;
   #SUBIR_CLAMPERS := #X114 AND NOT #STOP_ACT;
   #GRIPPERS := #X115 AND NOT #STOP_ACT;
   #CLAMPER := #X115 AND NOT #STOP_ACT;
   #MOVER_HOR := #X116 AND NOT #STOP_ACT;
   #Fin_Mantenimiento := #X117 AND NOT #STOP_ACT;


   //#Alarma_1 := (#Alarma_1 OR (#X31 AND #T1.Q)) AND NOT RESET_ALARMA;
   //#Alarma_2 := (#Alarma_2 OR (#X33 AND #T2.Q)) AND NOT RESET_ALARMA;

   //#Alarma := (#Alarma_1 OR #Alarma_2 OR #Alarma_3) AND NOT (#FORCE_INIT OR #RESET_ALARMA);
END_FUNCTION_BLOCK

FUNCTION_BLOCK "grafcet_120_vaciado_general"   // FB6, SCL
{ S7_Optimized_Access := 'TRUE' }
VERSION : 0.1
   VAR_INPUT
      Act_Vaciado : Bool;
      CI : Bool;
      Reset : Bool;
      Resume : Bool;
      fin_vac_1 : Bool;
      fin_vac_2 : Bool;
      fin_vac_3 : Bool;
      fin_sop_1 : Bool;
      fin_sop_2 : Bool;
      fin_sop_3 : Bool;
      fin_emb_1 : Bool;
      fin_emb_2 : Bool;
      fin_emb_3 : Bool;
      fin_emb_4 : Bool;
   END_VAR
   VAR_OUTPUT
      Vaciado_activado : Bool;
      act_vaciados_maquinas : Bool;
      Fin_vaciado : Bool;
   END_VAR
   VAR
      vac_finalizados : Bool;
      s120 : Bool;
      s121 : Bool;
      s122 : Bool;
      x120 : Bool;
      x121 : Bool;
      x122 : Bool;
      s120e : Bool;
      s121e : Bool;
      s122e : Bool;
      x120e : Bool;
      x121e : Bool;
      x122e : Bool;
      FORCE_CURRENT : Bool;
      FORCE_CURRENT_E : Bool;
      FORCE_INIT : Bool;
      FORCE_INIT_E : Bool;
   END_VAR
BEGIN
   //Flancos


   // EMERGENCIA
   #s120e := (#x122e AND #CI) OR "FirstScan";
   #s121e := #x120e AND FALSE;
   #s122e := #x121e;

   #x120e := #s120e OR (#x120e AND NOT #s121e);
   #x121e := #s121e OR (#x121e AND NOT #s122e);
   #x122e := #s122e OR (#x122e AND NOT #s120e);

   #FORCE_INIT_E := #x121e;
   #FORCE_CURRENT_E := #x122e;


   #FORCE_INIT := #FORCE_INIT_E;
   #FORCE_CURRENT := #FORCE_CURRENT_E ;


   #vac_finalizados := #fin_vac_1 AND #fin_vac_2 AND #fin_vac_3 AND #fin_sop_1 AND #fin_sop_2 AND #fin_sop_3 AND #fin_emb_1 AND #fin_emb_2 AND #fin_emb_3 AND #fin_emb_4;


   // PRODUCCIÓN
   #s120 := ("FirstScan" OR (#x122)) AND NOT #FORCE_CURRENT;
   #s121 := (#x120 AND (#Act_Vaciado)) AND NOT #FORCE_CURRENT;
   #s122 := (#x121 AND #vac_finalizados) AND NOT #FORCE_CURRENT;



   #x120 := (#s120 OR #x120 AND (NOT #s121)) OR #FORCE_INIT;
   #x121 := (#s121 OR #x121 AND (NOT #s122)) AND NOT #FORCE_INIT;
   #x122 := (#s122 OR #x122 AND (NOT #s120)) AND NOT #FORCE_INIT;

   #act_vaciados_maquinas := #x121;
   #Fin_vaciado := #x122;
END_FUNCTION_BLOCK

FUNCTION_BLOCK "grafcet_130_vaciados_maq"   // FB7, SCL
{ S7_Optimized_Access := 'TRUE' }
VERSION : 0.1
   VAR_INPUT
      Act_Vaciado_maquina : Bool;
      Fin_vaciado : Bool;
      CI : Bool;
   END_VAR
   VAR_OUTPUT
      Fin_vaciado_maq : Bool;
      Vaciados_maq_1 : Bool;
      Vaciados_maq_2 : Bool;
      Vaciados_maq_3 : Bool;
      Vaciados_maq_4 : Bool;
      Vaciados_maq_5 : Bool;
      Vaciados_maq_6 : Bool;
      Vaciados_maq_7 : Bool;
      Vaciados_maq_8 : Bool;
   END_VAR
   VAR
      S130 : Bool;
      S131 : Bool;
      s132 : Bool;
      x130 : Bool;
      x131 : Bool;
      x132 : Bool;
      s130e : Bool;
      s131e : Bool;
      s132e : Bool;
      x130e : Bool;
      x131e : Bool;
      x132e : Bool;
      FORCE_CURRENT : Bool;
      FORCE_CURRENT_E : Bool;
      FORCE_INIT : Bool;
      FORCE_INIT_E : Bool;
      T1 : TON_TIME;
   END_VAR
BEGIN
   //Flancos


   // EMERGENCIA
   #s130e := (#x132e AND #CI) OR "FirstScan";
   #s131e := #x130e AND FALSE;
   #s132e := #x131e;

   #x130e := #s130e OR (#x130e AND NOT #s131e);
   #x131e := #s131e OR (#x131e AND NOT #s132e);
   #x132e := #s132e OR (#x132e AND NOT #s130e);

   #FORCE_INIT_E := #x131e;
   #FORCE_CURRENT_E := #x132e;


   #FORCE_INIT := #FORCE_INIT_E ;
   #FORCE_CURRENT := #FORCE_CURRENT_E ;
   #T1(IN:=#x131,
       PT:=T#20s);




   // PRODUCCIÓN
   #S130 := ("FirstScan" OR (#x132 AND #Fin_vaciado )) AND NOT #FORCE_CURRENT;
   #S131 := (#x130 AND #Act_Vaciado_maquina) AND NOT #FORCE_CURRENT;
   #s132 := (#x131 AND #T1.Q) AND NOT #FORCE_CURRENT;



   #x130 := (#S130 OR #x130 AND (NOT #S131)) OR #FORCE_INIT;
   #x131 := (#S131 OR #x131 AND (NOT #s132)) AND NOT #FORCE_INIT;
   #x132 := (#s132 OR #x132 AND (NOT #S130)) AND NOT #FORCE_INIT;

   #Vaciados_maq_1 := #x131;
   #Vaciados_maq_2 := #x131;
   #Vaciados_maq_3 := #x131;
   #Vaciados_maq_4 := #x131;
   #Vaciados_maq_5 := #x131;
   #Vaciados_maq_6 := #x131;
   #Vaciados_maq_7 := #x131;
   #Vaciados_maq_8 := #x131;


   #Fin_vaciado_maq := #x132;
END_FUNCTION_BLOCK

FUNCTION_BLOCK "grafcet_125_vaciado_tipo1"   // FB8, SCL
{ S7_Optimized_Access := 'TRUE' }
VERSION : 0.1
   VAR_INPUT
      Act_Vaciado_Maquina : Bool;
      s2 : Bool;
      S3_2 : Bool;
      S3_3 : Bool;
      S3_1 : Bool;
      Fin_vaciado : Bool;
      CI : Bool;
   END_VAR
   VAR_OUTPUT
      QCINTA1 : Bool;
      QCINTA2 : Bool;
      QTrans : Bool;
      FIN_Vaciado_MAq : Bool;
   END_VAR
   VAR
      S125 : Bool;
      S126 : Bool;
      S126a : Bool;
      S126b : Bool;
      S127 : Bool;
      X125 : Bool;
      X126 : Bool;
      x126a : Bool;
      x126b : Bool;
      x127 : Bool;
      s1250e : Bool;
      s1251e : Bool;
      s1252e : Bool;
      x1250e : Bool;
      x1251e : Bool;
      x1252e : Bool;
      FORCE_INIT : Bool;
      FORCE_INIT_E : Bool;
      FORCE_CURRENT_E : Bool;
      S3 : Bool;
      T1 : TON_TIME;
      F_S2 : F_TRIG;
   END_VAR
BEGIN
   // EMERGENCIA
   #s1250e := (#x1252e AND #CI) OR "FirstScan";
   #s1251e := #x1250e AND FALSE;
   #s1252e := #x1251e;

   #x1250e := #s1250e OR (#x1250e AND NOT #s1251e);
   #x1251e := #s1251e OR (#x1251e AND NOT #s1252e);
   #x1252e := #s1252e OR (#x1252e AND NOT #s1250e);

   #FORCE_INIT_E := #x1251e;
   #FORCE_CURRENT_E := #x1252e;

   #S3 := #S3_1 OR #S3_2 OR #S3_3;

   #T1(IN:=#X126,
       PT:=T#10s);
   #F_S2(CLK:=#s2);



   // PRODUCCIÓN
   #S125 := ("FirstScan" OR (#x126b AND NOT #S3_1) OR (#x127 AND #Fin_vaciado)) AND NOT #FORCE_CURRENT_E;
   #S126 := ((#X125 AND #Act_Vaciado_Maquina) OR (#x126b AND NOT #S3)) AND NOT #FORCE_CURRENT_E;
   #S126a := (#X126 AND #F_S2.Q ) AND NOT #FORCE_CURRENT_E;
   #S126b := ((#X126 AND #S3) OR(#x126a AND #S3)  ) AND NOT #FORCE_CURRENT_E;
   #S127 := (#X126 AND #T1.Q) AND NOT #FORCE_CURRENT_E;

   // hay que revisar lo del FORCE_INIT
   #X125 := (#S125 OR #X125 AND NOT #S126) OR #FORCE_INIT_E;
   #X126 := (#S126 OR #X126 AND (NOT #S126a AND NOT #S127 AND NOT #S126b)) AND NOT #FORCE_INIT_E;
   #x126a := (#S126a OR #x126a AND NOT #S126b) AND NOT #FORCE_INIT_E;
   #x126b := (#S126b OR #x126b AND NOT #S125) AND NOT #FORCE_INIT_E;
   #x127 := (#S127 OR #x127 AND NOT #S125) AND NOT #FORCE_INIT_E;

   #QCINTA1 := #X126;
   #QCINTA2 := #X126 OR #x126a;
   #FIN_Vaciado_MAq := #x127;
   #QTrans := #x126b;
END_FUNCTION_BLOCK

FUNCTION_BLOCK "grafcet_140_manual_general"   // FB9, SCL
{ S7_Optimized_Access := 'TRUE' }
VERSION : 0.1
   VAR_INPUT
      act_manual : Bool;
      ci : Bool;
   END_VAR
   VAR_OUTPUT
      activar_manuales : Bool;
   END_VAR
   VAR
      s140 : Bool;
      s141 : Bool;
      s142 : Bool;
      x140 : Bool;
      x141 : Bool;
      s140e : Bool;
      s141e : Bool;
      s142e : Bool;
      x140e : Bool;
      x142e : Bool;
      x141e : Bool;
      FORCE_CURRENT : Bool;
      FORCE_INIT : Bool;
      FORCE_CURRENT_E : Bool;
      FORCE_INIT_E : Bool;
   END_VAR
BEGIN
   //Flancos


   // EMERGENCIA
   #s140e := (#x142e AND #ci) OR "FirstScan";
   #s141e := #x140e AND "Emergencia";
   #s142e := #x141e;

   #x140e := #s140e OR (#x140e AND NOT #s141e);
   #x141e := #s141e OR (#x141e AND NOT #s142e);
   #x142e := #s142e OR (#x142e AND NOT #s140e);

   #FORCE_INIT_E := #x141e;
   #FORCE_CURRENT_E := #x142e;


   #FORCE_INIT := #FORCE_INIT_E ;
   #FORCE_CURRENT := #FORCE_CURRENT_E ;



   // PRODUCCIÓN
   #s140 := ("FirstScan" OR (#x141 AND NOT #act_manual )) AND NOT #FORCE_CURRENT;
   #s141 := (#x140 AND #act_manual) AND NOT #FORCE_CURRENT;




   #x140 := (#s140 OR #x140 AND (NOT #s141)) OR #FORCE_INIT;
   #x141 := (#s141 OR #x141 AND (NOT #s140)) AND NOT #FORCE_INIT;


   #activar_manuales := #x141 AND NOT "Emergencia";
END_FUNCTION_BLOCK

FUNCTION_BLOCK "grafcet_145_manual_maquinas"   // FB10, SCL
{ S7_Optimized_Access := 'TRUE' }
VERSION : 0.1
   VAR_INPUT
      act_manual_maq : Bool;
      CI : Bool;
      Man_qc1 : Bool;
      man_qc2 : Bool;
      man_qc3 : Bool;
      man_qc4 : Bool;
      man_qtran1 : Bool;
      man_Qtran2 : Bool;
   END_VAR
   VAR_OUTPUT
      qcin1 : Bool;
      qcin2 : Bool;
      qcin3 : Bool;
      qcin4 : Bool;
      qtrans1 : Bool;
      qtrans2 : Bool;
   END_VAR
   VAR
      s145 : Bool;
      s146 : Bool;
      x145 : Bool;
      x146 : Bool;
      s145e : Bool;
      s146e : Bool;
      s147e : Bool;
      x145e : Bool;
      x146e : Bool;
      x147e : Bool;
      force_init : Bool;
      force_current : Bool;
      force_init_e : Bool;
      force_current_e : Bool;
   END_VAR
BEGIN
   //Flancos


   // EMERGENCIA
   #s145e := (#x147e AND #CI) OR "FirstScan";
   #s146e := #x145e AND "Emergencia";
   #s147e := #x146e;

   #x145e := #s145e OR (#x145e AND NOT #s146e);
   #x146e := #s146e OR (#x146e AND NOT #s147e);
   #x147e := #s147e OR (#x147e AND NOT #s145e);

   #force_init_e := #x146e;
   #force_current_e := #x147e;


   #force_init := #force_init_e ;
   #force_current := #force_current_e ;



   // PRODUCCIÓN
   #s145 := ("FirstScan" OR (#x146 AND NOT #act_manual_maq )) AND NOT #force_current;
   #s146 := (#x145 AND #act_manual_maq) AND NOT #force_current;




   #x145 := (#s145 OR #x145 AND (NOT #s146)) OR #force_init;
   #x146 := (#s146 OR #x146 AND (NOT #s145)) AND NOT #force_init;


   #qcin1 := (#x146 AND #Man_qc1) AND NOT "Emergencia";
   #qcin2 := (#x146 AND #man_qc2) AND NOT "Emergencia";
   #qcin3 := (#x146 AND #man_qc3) AND NOT "Emergencia";
   #qcin4 := (#x146 AND #man_qc4) AND NOT "Emergencia";
   #qtrans1 := (#x146 AND #man_qtran1) AND NOT "Emergencia";
   #qtrans2 := (#x146 AND #man_Qtran2) AND NOT "Emergencia";
END_FUNCTION_BLOCK

FUNCTION_BLOCK "Grafcet_1000_Emergencia"   // FB14, SCL
{ S7_Optimized_Access := 'TRUE' }
VERSION : 0.1
   VAR_INPUT
      "E" : Bool;
      REARME : Bool;
      Fin_Vaciado : Bool;
      Fin_Mantenimiento : Bool;
   END_VAR
   VAR_OUTPUT
      Emergencia : Bool;
      Activar_Vaciado : Bool;
      Activar_Mantenimiento : Bool;
   END_VAR
   VAR
      S1000 : Bool;
      S1001 : Bool;
      S1002 : Bool;
      S1003 : Bool;
      X1000 : Bool;
      X1001 : Bool;
      X1002 : Bool;
      X1003 : Bool;
      SETA : Bool;
   END_VAR
BEGIN

   #SETA := #E;

   #S1000 := "FirstScan" OR (#X1003 AND #Fin_Mantenimiento);
   #S1001 := #X1000 AND #SETA;
   #S1002 := #X1001 AND (NOT #SETA AND #REARME);
   #S1003 := #X1002 AND #Fin_Vaciado;

   #X1000 := #S1000 OR (#X1000 AND NOT #S1001);
   #X1001 := #S1001 OR (#X1001 AND NOT #S1002);
   #X1002 := #S1002 OR (#X1002 AND NOT #S1003);
   #X1003 := #S1003 OR (#X1003 AND NOT #S1000);


   #Emergencia := #X1001;
   #Activar_Vaciado := #X1002;
   #Activar_Mantenimiento := #X1003;
END_FUNCTION_BLOCK

FUNCTION_BLOCK "Grafcet_10_Final"   // FB25, SCL
{ S7_Optimized_Access := 'TRUE' }
VERSION : 0.1
   VAR_INPUT
      Act_Maquina : Bool;
      S_Pres : Bool;
      S1 : Bool;
      Sig_Maq_Libre : Bool;
      Mantenimiento_Cintas : Bool;
      Vaciado_cinta : Bool;
      Pieza_Rec : Bool;
      Reset : Bool;
      Resume : Bool;
      CI : Bool;
      Emergencia : Bool;
   END_VAR
   VAR_OUTPUT
      Emisor : Bool;
      Emisor_2 : Bool;
      Maq_Libre : Bool;
      QC1 : Bool;
      Act_SIG_MAQ : Bool;
      Alarma_Maquina : Bool;
      EstadoMaquina : Int;
   END_VAR
   VAR_IN_OUT
      Alarma_1 : Bool;
      Alarma_2 : Bool;
   END_VAR
   VAR
      S10 : Bool;
      S11 : Bool;
      S12 : Bool;
      S13 : Bool;
      S14 : Bool;
      S15 : Bool;
      X10 : Bool;
      X15 : Bool;
      X11 : Bool;
      X12 : Bool;
      X13 : Bool;
      X14 : Bool;
      S10e : Bool;
      S11e : Bool;
      S12e : Bool;
      X10e : Bool;
      X11e : Bool;
      X12e : Bool;
      FORCE_INIT : Bool;
      FORCE_INIT_E : Bool;
      FORCE_CURRENT_E : Bool;
      S10a : Bool;
      S11a : Bool;
      S12a : Bool;
      S13a : Bool;
      X10a : Bool;
      X11a : Bool;
      X12a : Bool;
      X13a : Bool;
      FORCE_CURRENT : Bool;
      STOP_ACT : Bool;
      RESET_ALARMA : Bool;
      Alarma : Bool;
      S11b : Bool;
      X11b : Bool;
      T1a : TON_TIME;
      trig_PR : R_TRIG;
   END_VAR
BEGIN
   //Flancos


   // EMERGENCIA
   #S10e := (#X12e AND #CI) OR "FirstScan";
   #S11e := #X10e AND "Emergencia";
   #S12e := #X11e;

   #X10e := #S10e OR (#X10e AND NOT #S11e);
   #X11e := #S11e OR (#X11e AND NOT #S12e);
   #X12e := #S12e OR (#X12e AND NOT #S10e);

   #FORCE_INIT_E := #X11e;
   #FORCE_CURRENT_E := #X12e;


   // ALARMAS
   #S10a := (#X13a AND NOT #FORCE_CURRENT_E) OR "FirstScan";
   #S11a := (#X10a AND #Alarma) AND NOT #FORCE_CURRENT_E;
   #S12a := (#X11a AND #Reset) AND NOT #FORCE_CURRENT_E;
   #S13a := (#X12a OR (#X11a AND #Resume)) AND NOT #FORCE_CURRENT_E;

   #X10a := #S10a OR (#X10a AND NOT #S11a) OR #FORCE_INIT_E;
   #X11a := (#S11a OR (#X11a AND NOT #S12a AND NOT #S13a)) AND NOT #FORCE_INIT_E;
   #X12a := (#S12a OR (#X12a AND NOT #S13a)) AND NOT #FORCE_INIT_E;
   #X13a := (#S13a OR (#X13a AND NOT #S10a)) AND NOT #FORCE_INIT_E;

   #STOP_ACT := #X11a;
   #FORCE_INIT := #FORCE_INIT_E OR #X12a;
   #FORCE_CURRENT := #FORCE_CURRENT_E OR #X11a;
   #RESET_ALARMA := #X13a;

   #trig_PR(CLK:=#Pieza_Rec);

   // PRODUCCIÓN
   #S10 := "FirstScan" OR( (#X15 AND #trig_PR.Q)) AND NOT #FORCE_CURRENT;
   #S11 := (#X10 AND #Act_Maquina) AND NOT #FORCE_CURRENT;
   #S11b := (#X11 AND #S_Pres ) AND NOT #FORCE_CURRENT;
   #S12 := (#X11b AND( NOT #S_Pres )) AND NOT #FORCE_CURRENT;
   #S13 := (#X12 AND #S1) AND NOT #FORCE_CURRENT;
   #S14 := (#X13 AND #Sig_Maq_Libre) AND NOT #FORCE_CURRENT;
   #S15 := (#X14 AND NOT #S1) AND NOT #FORCE_CURRENT;


   #X10 := (#S10 OR #X10 AND (NOT #S11)) OR #FORCE_INIT;
   #X11 := (#S11 OR #X11 AND (NOT #S11b)) AND NOT #FORCE_INIT;
   #X11b := (#S11b OR #X11b AND (NOT #S12)) AND NOT #FORCE_INIT;
   #X12 := (#S12 OR #X12 AND (NOT #S13 AND NOT #S14)) AND NOT #FORCE_INIT;
   #X13 := (#S13 OR #X13 AND (NOT #S14)) AND NOT #FORCE_INIT;
   #X14 := (#S14 OR #X14 AND (NOT #S15)) AND NOT #FORCE_INIT;
   #X15 := (#S15 OR #X15 AND (NOT #S10)) AND NOT #FORCE_INIT;


   #Maq_Libre := #X10 AND NOT #STOP_ACT;
   #Emisor_2 := (#X11 AND NOT #S_Pres) AND NOT #STOP_ACT;
   #Emisor := (#X11 AND NOT #S_Pres) AND NOT #STOP_ACT;
   #QC1 := (#X11 OR #X11b OR  #X12 OR #X14 OR #Mantenimiento_Cintas OR #Vaciado_cinta)  AND NOT #STOP_ACT;
   #Act_SIG_MAQ := #X14 AND NOT #STOP_ACT;


   #T1a(IN:=#X12,
        PT:=T#10s);
   //#Alarma_1 := #Alarma_1 OR (#X12 AND #S_Pres)AND NOT #RESET_ALARMA;
   #Alarma_2 := #Alarma_2 OR (#T1a.Q) AND NOT #RESET_ALARMA;
   #Alarma := (#Alarma_1 OR #Alarma_2) AND NOT (#FORCE_INIT OR #RESET_ALARMA);
   #Alarma_Maquina := #Alarma;

   IF #X10 = TRUE AND NOT #Alarma AND NOT "Emergencia" THEN
       #EstadoMaquina := 0;
   END_IF;
   IF #X10 = FALSE AND NOT #Alarma AND NOT "Emergencia" THEN
       #EstadoMaquina := 1;
   END_IF;
   IF #Alarma AND NOT "Emergencia" THEN
       #EstadoMaquina := 2;
   END_IF;
   IF "Emergencia" THEN
       #EstadoMaquina := 3;
   END_IF;
END_FUNCTION_BLOCK

FUNCTION_BLOCK "Grafcet_20_FInal"   // FB26, SCL
{ S7_Optimized_Access := 'TRUE' }
VERSION : 0.1
   VAR_INPUT
      Act_Proceso : Bool;
      SigMaqLibre : Bool;
      SA_Bueno : Bool;
      SA_Malo : Bool;
      SB : Bool;
      Mantenimiento_Cintas : Bool;
      Mantenimiento_Transfes : Bool;
      vaciado_cinta : Bool;
      vaciado_Trans : Bool;
      CI : Bool;
      Reset : Bool;
      Resume : Bool;
   END_VAR
   VAR_OUTPUT
      Maq_Libre : Bool;
      QC2 : Bool;
      QTRANS : Bool;
      Act_SIG_MAQ_Buena : Bool;
      Act_SIG_MAQ_Mala : Bool;
      TipoAbuena : Bool;
      TipoAMala : Bool;
      TipoB : Bool;
      Alarma_Maquina : Bool;
      Pieza_Rec : Bool;
   END_VAR
   VAR_IN_OUT
      Alarma_1 : Bool;
      Alarma_2 : Bool;
   END_VAR
   VAR
      S20 : Bool;
      S21 : Bool;
      S22 : Bool;
      S23 : Bool;
      S24 : Bool;
      S22b : Bool;
      S23b : Bool;
      X20 : Bool;
      X21 : Bool;
      X22 : Bool;
      X22b : Bool;
      X23 : Bool;
      X23b : Bool;
      X24 : Bool;
      S20a : Bool;
      S21a : Bool;
      S22a : Bool;
      S23a : Bool;
      X20a : Bool;
      X21a : Bool;
      X22a : Bool;
      X23a : Bool;
      S20e : Bool;
      S21e : Bool;
      S22e : Bool;
      X20e : Bool;
      X21e : Bool;
      X22e : Bool;
      FORCE_INIT : Bool;
      FORCE_INIT_E : Bool;
      FORCE_CURRENT : Bool;
      FORCE_CURRENT_E : Bool;
      STOP_ACT : Bool;
      RESET_ALARMA : Bool;
      Alarma : Bool;
      T1 : TON_TIME;
      T1a : TON_TIME;
      T2a : TON_TIME;
   END_VAR
BEGIN

   // EMERGENCIA
   #S20e := (#X22e AND #CI) OR "FirstScan";
   #S21e := #X20e AND "Emergencia";
   #S22e := #X21e;

   #X20e := #S20e OR (#X20e AND NOT #S21e);
   #X21e := #S21e OR (#X21e AND NOT #S22e);
   #X22e := #S22e OR (#X22e AND NOT #S20e);

   #FORCE_INIT_E := #X21e;
   #FORCE_CURRENT_E := #X22e;


   // ALARMAS
   #S20a := (#X23a AND NOT #FORCE_CURRENT_E) OR "FirstScan";
   #S21a := (#X20a AND #Alarma) AND NOT #FORCE_CURRENT_E;
   #S22a := (#X21a AND #Reset) AND NOT #FORCE_CURRENT_E;
   #S23a := (#X22a OR (#X21a AND #Resume)) AND NOT #FORCE_CURRENT_E;

   #X20a := #S20a OR (#X20a AND NOT #S21a) OR #FORCE_INIT_E;
   #X21a := (#S21a OR (#X21a AND NOT #S22a AND NOT #S23a)) AND NOT #FORCE_INIT_E;
   #X22a := (#S22a OR (#X22a AND NOT #S23a)) AND NOT #FORCE_INIT_E;
   #X23a := (#S23a OR (#X23a AND NOT #S20a)) AND NOT #FORCE_INIT_E;

   #STOP_ACT := #X21a;
   #FORCE_INIT := #FORCE_INIT_E OR #X22a;
   #FORCE_CURRENT := #FORCE_CURRENT_E OR #X21a;
   #RESET_ALARMA := #X23a;
   #T1(IN:=#X24,
       PT:=T#2s);




   // PRODUCCIÓN
   #S20 := ("FirstScan" OR (#X22b AND NOT #SA_Bueno) OR (#X23b AND NOT #SA_Malo) OR (#X24 AND #T1.Q) ) AND NOT #FORCE_CURRENT;
   #S21 := (#X20 AND #Act_Proceso) AND NOT #FORCE_CURRENT;
   #S22 := (#X21 AND #SA_Bueno) AND NOT #FORCE_CURRENT;
   #S22b := (#X22 AND #SigMaqLibre) AND NOT #FORCE_CURRENT;
   #S23 := (#X21 AND #SA_Malo AND NOT #SA_Bueno) AND NOT #FORCE_CURRENT;
   #S23b := (#X23 AND #SigMaqLibre) AND NOT #FORCE_CURRENT;
   #S24 := (#X21 AND #SB) AND NOT #FORCE_CURRENT;



   #X20 := (#S20 OR #X20 AND (NOT #S21)) OR #FORCE_INIT;
   #X21 := (#S21 OR #X21 AND (NOT #S22 AND NOT #S23 AND NOT #S24)) AND NOT #FORCE_INIT;
   #X22 := (#S22 OR #X22 AND (NOT #S22b)) AND NOT #FORCE_INIT;
   #X22b := (#S22b OR #X22b AND (NOT #S20)) AND NOT #FORCE_INIT;
   #X23 := (#S23 OR #X23 AND (NOT #S23b)) AND NOT #FORCE_INIT;
   #X23b := (#S23b OR #X23b AND (NOT #S20)) AND NOT #FORCE_INIT;
   #X24 := (#S24 OR #X24 AND (NOT #S20)) AND NOT #FORCE_INIT;



   #Maq_Libre := #X20 AND NOT #STOP_ACT;
   #QC2 := (#X21 OR #X22b OR #X23b OR #Mantenimiento_Cintas OR #vaciado_cinta) AND NOT #STOP_ACT;
   #QTRANS := (#X24 OR #Mantenimiento_Transfes OR #vaciado_Trans) AND NOT #STOP_ACT;
   #Act_SIG_MAQ_Buena := #X22b AND NOT #STOP_ACT;
   #Act_SIG_MAQ_Mala := #X23b AND NOT #STOP_ACT;
   #Pieza_Rec := (#X22 OR #X23 OR #X24) AND NOT #STOP_ACT;

   #TipoAbuena := #X22b;
   #TipoAMala := #X23b;
   #TipoB := #X24;

   #T1a(IN := #X21,
        PT := T#10s);
   #T2a(IN := #X22b OR #X23b,
        PT := T#5s);


   #Alarma_1 := (#Alarma_1 OR (#T1a.Q)) AND NOT #RESET_ALARMA;
   //#Alarma_2 := (#Alarma_2 OR (#T2a.Q)) AND NOT #RESET_ALARMA;

   #Alarma := (#Alarma_1 OR #Alarma_2) AND NOT (#FORCE_INIT OR #RESET_ALARMA);
   #Alarma_Maquina := #Alarma;
END_FUNCTION_BLOCK

FUNCTION_BLOCK "grafcet_30_fina"   // FB27, SCL
{ S7_Optimized_Access := 'TRUE' }
VERSION : 0.1
   VAR_INPUT
      Act_Proceso_Bueno : Bool;
      Act_Proceso_malo : Bool;
      S3 : Bool;
      SigMaqLibre : Bool;
      Mantenimiento_Cinta : Bool;
      vaciado_cinta : Bool;
      Reset : Bool;
      Resume : Bool;
      CI : Bool;
   END_VAR
   VAR_OUTPUT
      Maq_Libre : Bool;
      QC3 : Bool;
      Act_SIG_MAQ_Buena : Bool;
      Act_SIG_MAQ_Mala : Bool;
      Alarma_Maquina : Bool;
   END_VAR
   VAR_IN_OUT
      Alarma_1 : Bool;
      Alarma_2 : Bool;
   END_VAR
   VAR
      S30 : Bool;
      S31 : Bool;
      S31b : Bool;
      S31c : Bool;
      S32 : Bool;
      S32b : Bool;
      S32c : Bool;
      X30 : Bool;
      X31 : Bool;
      X32 : Bool;
      X32b : Bool;
      X32c : Bool;
      X31b : Bool;
      X31c : Bool;
      S30e : Bool;
      S31e : Bool;
      S32e : Bool;
      X30e : Bool;
      X31e : Bool;
      X32e : Bool;
      X30a : Bool;
      X31a : Bool;
      X32a : Bool;
      X33a : Bool;
      S30a : Bool;
      S31a : Bool;
      S32a : Bool;
      S33a : Bool;
      FORCE_INIT_E : Bool;
      FORCE_INIT : Bool;
      FORCE_CURRENT_e : Bool;
      FORCE_CURRENT : Bool;
      RESET_ALARMA : Bool;
      STOP_ACT : Bool;
      Alarma : Bool;
      T1a : TON_TIME;
      T2a : TON_TIME;
   END_VAR
BEGIN
   //Flancos


   // EMERGENCIA
   #S30e := (#X32e AND #CI) OR "FirstScan";
   #S31e := #X30e AND "Emergencia";
   #S32e := #X31e;

   #X30e := #S30e OR (#X30e AND NOT #S31e);
   #X31e := #S31e OR (#X31e AND NOT #S32e);
   #X32e := #S32e OR (#X32e AND NOT #S30e);

   #FORCE_INIT_E := #X31e;
   #FORCE_CURRENT_e := #X32e;


   // ALARMAS
   #S30a := (#X33a AND NOT #FORCE_CURRENT_e) OR "FirstScan";
   #S31a := (#X30a AND #Alarma) AND NOT #FORCE_CURRENT_e;
   #S32a := (#X31a AND #Reset) AND NOT #FORCE_CURRENT_e;
   #S33a := (#X32a OR (#X31a AND #Resume)) AND NOT #FORCE_CURRENT_e;

   #X30a := #S30a OR (#X30a AND NOT #S31a) OR #FORCE_INIT_E;
   #X31a := (#S31a OR (#X31a AND NOT #S32a AND NOT #S33a)) AND NOT #FORCE_INIT_E;
   #X32a := (#S32a OR (#X32a AND NOT #S33a)) AND NOT #FORCE_INIT_E;
   #X33a := (#S33a OR (#X33a AND NOT #S30a)) AND NOT #FORCE_INIT_E;

   #STOP_ACT := #X31a;
   #FORCE_INIT := #FORCE_INIT_E OR #X32a;
   #FORCE_CURRENT := #FORCE_CURRENT_e OR #X31a;
   #RESET_ALARMA := #X33a;


   // PRODUCCIÓN
   #S30 := ("FirstScan" OR (#X31c AND NOT #S3) OR (#X32c AND NOT #S3)) AND NOT #FORCE_CURRENT;
   #S31 := (#X30 AND #Act_Proceso_Bueno) AND NOT #FORCE_CURRENT;
   #S31b := (#X31 AND #S3) AND NOT #FORCE_CURRENT;
   #S31c := (#X31b AND #SigMaqLibre) AND NOT #FORCE_CURRENT;
   #S32 := (#X30 AND #Act_Proceso_malo) AND NOT #FORCE_CURRENT;
   #S32b := (#X32 AND #S3) AND NOT #FORCE_CURRENT;
   #S32c := (#X32b AND #SigMaqLibre) AND NOT #FORCE_CURRENT;



   #X30 := (#S30 OR #X30 AND (NOT #S31 AND NOT #S32)) OR #FORCE_INIT;
   #X31 := (#S31 OR #X31 AND (NOT #S31b)) AND NOT #FORCE_INIT;
   #X31b := (#S31b OR #X31b AND (NOT #S31c)) AND NOT #FORCE_INIT;
   #X31c := (#S31c OR #X31c AND (NOT #S30)) AND NOT #FORCE_INIT;
   #X32 := (#S32 OR #X32 AND (NOT #S32b)) AND NOT #FORCE_INIT;
   #X32b := (#S32b OR #X32b AND (NOT #S32c)) AND NOT #FORCE_INIT;
   #X32c := (#S32c OR #X32c AND (NOT #S30)) AND NOT #FORCE_INIT;



   #Maq_Libre := #X30 AND NOT #STOP_ACT;
   #QC3 := (#X31 OR #X31c OR #X32 OR #X32c OR #Mantenimiento_Cinta OR #vaciado_cinta) AND NOT #STOP_ACT;
   #Act_SIG_MAQ_Buena := #X31c AND NOT #STOP_ACT;
   #Act_SIG_MAQ_Mala := #X32c AND NOT #STOP_ACT;

   #T1a(IN:=#X31 OR #X32,
        PT:=T#5s);
   #T2a(IN := #X31c OR #X32c,
        PT := T#5s);


   //#Alarma_1 := (#Alarma_1 OR (#T1a.Q)) AND NOT #RESET_ALARMA;
   //#Alarma_2 := (#Alarma_2 OR (#T2a.Q)) AND NOT #RESET_ALARMA;

   //#Alarma := (#Alarma_1 OR #Alarma_2 ) AND NOT (#FORCE_INIT OR #RESET_ALARMA);
   //#Alarma_Maquina := #Alarma;
END_FUNCTION_BLOCK

FUNCTION_BLOCK "grafcet_40_final"   // FB28, SCL
{ S7_Optimized_Access := 'TRUE' }
VERSION : 0.1
   VAR_INPUT
      Act_Proceso_Bueno : Bool;
      Act_Proceso_Malo : Bool;
      S4 : Bool;
      SigMaqLibre : Bool;
      Mantenimiento_Cinta : Bool;
      Mantenimiento_Trans : Bool;
      vaciado_cinta : Bool;
      vaciado_Trans : Bool;
      CI : Bool;
      Reset : Bool;
      Resume : Bool;
   END_VAR
   VAR_OUTPUT
      Maq_Libre : Bool;
      QC4 : Bool;
      QTRANS : Bool;
      Act_Sig_Maq : Bool;
      Alarma_Maquina : Bool;
   END_VAR
   VAR_IN_OUT
      Alarma_1 : Bool;
      Alarma_2 : Bool;
      Alarma_3 : Bool;
   END_VAR
   VAR
      S40 : Bool;
      S41 : Bool;
      S42 : Bool;
      S41b : Bool;
      S41c : Bool;
      S42b : Bool;
      X40 : Bool;
      X41 : Bool;
      X41b : Bool;
      X41c : Bool;
      X42 : Bool;
      X42b : Bool;
      S40e : Bool;
      S41e : Bool;
      S42e : Bool;
      X40e : Bool;
      X41e : Bool;
      X42e : Bool;
      S40a : Bool;
      S41a : Bool;
      S42a : Bool;
      S43a : Bool;
      X40a : Bool;
      X41a : Bool;
      X42a : Bool;
      X43a : Bool;
      FORCE_CURRENT : Bool;
      FORCE_CURRENT_E : Bool;
      FORCE_INIT : Bool;
      FORCE_INIT_E : Bool;
      STOP_ACT : Bool;
      RESET_ALARMA : Bool;
      Alarma : Bool;
      T1a : TON_TIME;
      T2a : TON_TIME;
      T3a : TON_TIME;
   END_VAR
BEGIN


   // EMERGENCIA
   #S40e := (#X42e AND #CI) OR "FirstScan";
   #S41e := #X40e AND "Emergencia";
   #S42e := #X41e;

   #X40e := #S40e OR (#X40e AND NOT #S41e);
   #X41e := #S41e OR (#X41e AND NOT #S42e);
   #X42e := #S42e OR (#X42e AND NOT #S40e);

   #FORCE_INIT_E := #X41e;
   #FORCE_CURRENT_E := #X42e;


   // ALARMAS
   #S40a := (#X43a AND NOT #FORCE_CURRENT_E) OR "FirstScan";
   #S41a := (#X40a AND #STOP_ACT) AND NOT #FORCE_CURRENT_E;
   #S42a := (#X41a AND #Reset) AND NOT #FORCE_CURRENT_E;
   #S43a := (#X42a OR (#X41a AND #Resume)) AND NOT #FORCE_CURRENT_E;

   #X40a := #S40a OR (#X40a AND NOT #S41a) OR #FORCE_INIT_E;
   #X41a := (#S41a OR (#X41a AND NOT #S42a AND NOT #S43a)) AND NOT #FORCE_INIT_E;
   #X42a := (#S42a OR (#X42a AND NOT #S43a)) AND NOT #FORCE_INIT_E;
   #X43a := (#S43a OR (#X43a AND NOT #S40a)) AND NOT #FORCE_INIT_E;

   #STOP_ACT := #X41a;
   #FORCE_INIT := #FORCE_INIT_E OR #X42a;
   #FORCE_CURRENT := #FORCE_CURRENT_E OR #X41a;
   #RESET_ALARMA := #X43a;



   // PRODUCCIÓN
   #S40 := ("FirstScan" OR (#X41c AND NOT #S4) OR (#X42b AND NOT #S4)) AND NOT #FORCE_CURRENT;
   #S41 := (#X40 AND #Act_Proceso_Bueno) AND NOT #FORCE_CURRENT;
   #S41b := (#X41 AND #S4) AND NOT #FORCE_CURRENT;
   #S41c := (#X41b AND #SigMaqLibre) AND NOT #FORCE_CURRENT;
   #S42 := (#X40 AND #Act_Proceso_Malo) AND NOT #FORCE_CURRENT;
   #S42b := (#X42 AND #S4) AND NOT #FORCE_CURRENT;



   #X40 := (#S40 OR #X40 AND (NOT #S41 AND NOT #S42)) OR #FORCE_INIT;
   #X41 := (#S41 OR #X41 AND (NOT #S41b)) AND NOT #FORCE_INIT;
   #X41b := (#S41b OR #X41b AND (NOT #S41c)) AND NOT #FORCE_INIT;
   #X41c := (#S41c OR #X41c AND (NOT #S40)) AND NOT #FORCE_INIT;
   #X42 := (#S42 OR #X42 AND (NOT #S42b)) AND NOT #FORCE_INIT;
   #X42b := (#S42b OR #X42b AND (NOT #S40)) AND NOT #FORCE_INIT;



   #Maq_Libre := #X40 AND NOT #STOP_ACT;
   #QC4 := (#X41 OR #X41c OR #X42 OR #Mantenimiento_Cinta OR #vaciado_cinta) AND NOT #STOP_ACT;
   #Act_Sig_Maq := #X41c AND NOT #STOP_ACT;
   #QTRANS := (#X42b OR #Mantenimiento_Trans OR #vaciado_Trans) AND NOT #STOP_ACT;

   #T1a(IN:=#X41 OR #X42,
        PT:=T#5s);
   #T2a(IN := #X41c,
        PT := T#5s);
   #T3a(IN := #X42b,
        PT := T#5s);


   //#Alarma_1 := (#Alarma_1 OR #T1a.Q) AND NOT #RESET_ALARMA;
   //#Alarma_2 := (#Alarma_2 OR #T2a.Q) AND NOT #RESET_ALARMA;
   //#Alarma_3 := (#Alarma_3 OR #T3a.Q) AND NOT #RESET_ALARMA;

   //#Alarma := (#Alarma_1 OR #Alarma_2 OR #Alarma_3) AND NOT (#FORCE_INIT OR #RESET_ALARMA);
END_FUNCTION_BLOCK

FUNCTION_BLOCK "grafcet_50_Final"   // FB29, SCL
{ S7_Optimized_Access := 'TRUE' }
VERSION : 0.1
   VAR_INPUT
      Act_Proceso : Bool;
      S5 : Bool;
      HaySoporte : Bool;
      CI : Bool;
      Mantenimiento_Cinta : Bool;
      Mantenimiento_Clamper : Bool;
      Mantenimiento_Gripper : Bool;
      Mantenimiento_BajarGripper : Bool;
      Mantenimiento_MOVHOR : Bool;
      vaciado_cinta : Bool;
      vaciado_subclamper : Bool;
      Reset : Bool;
      Resume : Bool;
   END_VAR
   VAR_OUTPUT
      Maq_Libre : Bool;
      QC5 : Bool;
      QC6 : Bool;
      QC7 : Bool;
      QCLAMP : Bool;
      qsubclamp : Bool;
      QBAJ : Bool;
      QGRIPPER : Bool;
      QHOR : Bool;
      HayPieza : Bool;
      Pieza_Empaquetada : Bool;
      Alarma_Maquina : Bool;
   END_VAR
   VAR_IN_OUT
      Alarma_1 : Bool;
   END_VAR
   VAR
      S50 : Bool;
      S51 : Bool;
      S52 : Bool;
      S53 : Bool;
      S54 : Bool;
      S55 : Bool;
      S56 : Bool;
      S57 : Bool;
      S58 : Bool;
      S59 : Bool;
      S60 : Bool;
      S61 : Bool;
      S62 : Bool;
      X50 : Bool;
      X51 : Bool;
      X52 : Bool;
      X53 : Bool;
      X54 : Bool;
      X55 : Bool;
      X56 : Bool;
      X57 : Bool;
      X58 : Bool;
      X59 : Bool;
      X60 : Bool;
      X61 : Bool;
      X62 : Bool;
      S50e : Bool;
      S51e : Bool;
      S52e : Bool;
      X50e : Bool;
      X51e : Bool;
      X52e : Bool;
      S50a : Bool;
      S51a : Bool;
      S52a : Bool;
      S53a : Bool;
      X50a : Bool;
      X51a : Bool;
      X52a : Bool;
      X53a : Bool;
      FORCE_INIT : Bool;
      FORCE_INIT_E : Bool;
      FORCE_CURRENT : Bool;
      FORCE_CURRENT_E : Bool;
      STOP_ACT : Bool;
      RESET_ALARMA : Bool;
      Alarma : Bool;
      T1 : TON_TIME;
      T2 : TON_TIME;
      T3 : TON_TIME;
      T4 : TON_TIME;
      T5 : TON_TIME;
      T6 : TON_TIME;
      T7 : TON_TIME;
      T8 : TON_TIME;
      T9 : TON_TIME;
      T1a : TON_TIME;
   END_VAR
BEGIN


   // EMERGENCIA
   #S50e := (#X52e AND #CI) OR "FirstScan";
   #S51e := #X50e AND "Emergencia";
   #S52e := #X51e;

   #X50e := #S50e OR (#X50e AND NOT #S51e);
   #X51e := #S51e OR (#X51e AND NOT #S52e);
   #X52e := #S52e OR (#X52e AND NOT #S50e);

   #FORCE_INIT_E := #X51e;
   #FORCE_CURRENT_E := #X52e;


   // ALARMAS
   #S50a := (#X53a AND NOT #FORCE_CURRENT_E) OR "FirstScan";
   #S51a := (#X50a AND #Alarma) AND NOT #FORCE_CURRENT_E;
   #S52a := (#X51a AND #Reset) AND NOT #FORCE_CURRENT_E;
   #S53a := (#X52a OR (#X51a AND #Resume)) AND NOT #FORCE_CURRENT_E;

   #X50a := #S50a OR (#X50a AND NOT #S51a) OR #FORCE_INIT_E;
   #X51a := (#S51a OR (#X51a AND NOT #S52a AND NOT #S53a)) AND NOT #FORCE_INIT_E;
   #X52a := (#S52a OR (#X52a AND NOT #S53a)) AND NOT #FORCE_INIT_E;
   #X53a := (#S53a OR (#X53a AND NOT #S50a)) AND NOT #FORCE_INIT_E;

   #STOP_ACT := #X51a;
   #FORCE_INIT := #FORCE_INIT_E OR #X52a;
   #FORCE_CURRENT := #FORCE_CURRENT_E OR #X51a;
   #RESET_ALARMA := #X53a;

   #T1(IN:=#X52,
       PT:=T#2s);
   #T2(IN := #X53,
       PT := T#2s);
   #T3(IN := #X55,
       PT := T#2s);
   #T4(IN := #X56,
       PT := T#2s);
   #T5(IN := #X57,
       PT := T#2s);
   #T6(IN := #X58,
       PT := T#2s);
   #T7(IN := #X59,
       PT := T#2s);
   #T8(IN := #X60,
       PT := T#2s);
   #T9(IN := #X61,
       PT := T#2s);



   // PRODUCCIÓN
   #S50 := ("FirstScan" OR (#X62)) AND NOT #FORCE_CURRENT;
   #S51 := (#X50 AND #Act_Proceso) AND NOT #FORCE_CURRENT;
   #S52 := (#X51 AND #S5) AND NOT #FORCE_CURRENT;
   #S53 := (#X52 AND #T1.Q) AND NOT #FORCE_CURRENT;
   #S54 := (#X53 AND #T2.Q) AND NOT #FORCE_CURRENT;
   #S55 := (#X54 AND #HaySoporte) AND NOT #FORCE_CURRENT;
   #S56 := (#X55 AND #T3.Q) AND NOT #FORCE_CURRENT;
   #S57 := (#X56 AND #T4.Q) AND NOT #FORCE_CURRENT;
   #S58 := (#X57 AND #T5.Q) AND NOT #FORCE_CURRENT;
   #S59 := (#X58 AND #T6.Q) AND NOT #FORCE_CURRENT;
   #S60 := (#X59 AND #T7.Q) AND NOT #FORCE_CURRENT;
   #S61 := (#X60 AND #T8.Q) AND NOT #FORCE_CURRENT;
   #S62 := (#X61 AND #T9.Q) AND NOT #FORCE_CURRENT;


   #X50 := (#S50 OR #X50 AND (NOT #S51)) OR #FORCE_INIT;
   #X51 := (#S51 OR #X51 AND (NOT #S52)) AND NOT #FORCE_INIT;
   #X52 := (#S52 OR #X52 AND (NOT #S53)) AND NOT #FORCE_INIT;
   #X53 := (#S53 OR #X53 AND (NOT #S54)) AND NOT #FORCE_INIT;
   #X54 := (#S54 OR #X54 AND (NOT #S55)) AND NOT #FORCE_INIT;
   #X55 := (#S55 OR #X55 AND (NOT #S56)) AND NOT #FORCE_INIT;
   #X56 := (#S56 OR #X56 AND (NOT #S57)) AND NOT #FORCE_INIT;
   #X57 := (#S57 OR #X57 AND (NOT #S58)) AND NOT #FORCE_INIT;
   #X58 := (#S58 OR #X58 AND (NOT #S59)) AND NOT #FORCE_INIT;
   #X59 := (#S59 OR #X59 AND (NOT #S60)) AND NOT #FORCE_INIT;
   #X60 := (#S60 OR #X60 AND (NOT #S61)) AND NOT #FORCE_INIT;
   #X61 := (#S61 OR #X61 AND (NOT #S62)) AND NOT #FORCE_INIT;
   #X62 := (#S62 OR #X62 AND (NOT #S50)) AND NOT #FORCE_INIT;



   #Maq_Libre := #X50 AND NOT #STOP_ACT;
   #QC5 := (#X51 OR #X52 OR #Mantenimiento_Cinta OR #vaciado_cinta) AND NOT #STOP_ACT;
   #QC6 := (#X51 OR #X52 OR #Mantenimiento_Cinta OR #vaciado_cinta) AND NOT #STOP_ACT;
   #QC7 := (#X51 OR #X52 OR #X53 OR #X54 OR #Mantenimiento_Cinta OR #vaciado_cinta) AND NOT #STOP_ACT;
   #QCLAMP := (#X53 OR #X54 OR #X55 OR #X56 OR #X57 OR #Mantenimiento_Clamper)AND NOT #STOP_ACT;
   #QBAJ := (#X55 OR #X56 OR #X59 OR #X60 OR #Mantenimiento_BajarGripper) AND NOT #STOP_ACT;
   #QGRIPPER := (#X56 OR #X57 OR #X58 OR #X59 OR #Mantenimiento_Gripper) AND NOT #STOP_ACT;
   #QHOR := (#X58 OR #X59 OR #X60 OR #X61 OR #Mantenimiento_MOVHOR) AND NOT #STOP_ACT;
   #qsubclamp := #vaciado_subclamper AND NOT #STOP_ACT;
   #HayPieza := #X54 AND NOT #STOP_ACT;
   #Pieza_Empaquetada := #X62 AND NOT #STOP_ACT;


   #T1a(IN:=#X51,
        PT:=T#20s);


   //#Alarma_1 := (#Alarma_1 OR (#T1a.Q)) AND NOT #RESET_ALARMA;

   //#Alarma := (#Alarma_1) AND NOT (#FORCE_INIT OR #RESET_ALARMA);
   //#Alarma_Maquina := #Alarma;
END_FUNCTION_BLOCK

FUNCTION_BLOCK "Grafcet_70_Final"   // FB30, SCL
{ S7_Optimized_Access := 'TRUE' }
VERSION : 0.1
   VAR_INPUT
      Act_Proceso : Bool;
      S5 : Bool;
      Pieza_Empaquetada : Bool;
      SigMaqLibre : Bool;
      Mantenimiento_Cinta : Bool;
      Mantenimiento_Clamper : Bool;
      Mantenimiento_SubirClamp : Bool;
      vaciado_cinta : Bool;
      vaciado_subclamp : Bool;
      CI : Bool;
      Reset : Bool;
      Resume : Bool;
   END_VAR
   VAR_OUTPUT
      Maq_Libre : Bool;
      QC5 : Bool;
      QC6 : Bool;
      QC7 : Bool;
      QCLAMP : Bool;
      QCLAMP_SUB : Bool;
      Act_SIG_MAQ : Bool;
      HayPieza : Bool;
      Alarma_Maquina : Bool;
   END_VAR
   VAR_IN_OUT
      Alarma_1 : Bool;
   END_VAR
   VAR
      S70 : Bool;
      S71 : Bool;
      S72 : Bool;
      S73 : Bool;
      S74 : Bool;
      S75 : Bool;
      S76 : Bool;
      X70 : Bool;
      X71 : Bool;
      X72 : Bool;
      X73 : Bool;
      X74 : Bool;
      X75 : Bool;
      X76 : Bool;
      S70e : Bool;
      S71e : Bool;
      S72e : Bool;
      X70e : Bool;
      X71e : Bool;
      X72e : Bool;
      X70a : Bool;
      X71a : Bool;
      X72a : Bool;
      X73a : Bool;
      S70a : Bool;
      S71a : Bool;
      S72a : Bool;
      S73a : Bool;
      STOP_ACT : Bool;
      FORCE_INIT : Bool;
      FORCE_INIT_E : Bool;
      FORCE_CURRENT : Bool;
      FORCE_CURRENT_E : Bool;
      RESET_ALARMA : Bool;
      Alarma : Bool;
      T1 : TON_TIME;
      T2 : TON_TIME;
      T3 : TON_TIME;
      T1a : TON_TIME;
   END_VAR
BEGIN
   //Flancos


   // EMERGENCIA
   #S70e := (#X72e AND #CI) OR "FirstScan";
   #S71e := #X70e AND "Emergencia";
   #S72e := #X71e;

   #X70e := #S70e OR (#X70e AND NOT #S71e);
   #X71e := #S71e OR (#X71e AND NOT #S72e);
   #X72e := #S72e OR (#X72e AND NOT #S70e);

   #FORCE_INIT_E := #X71e;
   #FORCE_CURRENT_E := #X72e;


   // ALARMAS
   #S70a := (#X73a AND NOT #FORCE_CURRENT_E) OR "FirstScan";
   #S71a := (#X70a AND #Alarma) AND NOT #FORCE_CURRENT_E;
   #S72a := (#X71a AND #Reset) AND NOT #FORCE_CURRENT_E;
   #S73a := (#X72a OR (#X71a AND #Resume)) AND NOT #FORCE_CURRENT_E;

   #X70a := #S70a OR (#X70a AND NOT #S71a) OR #FORCE_INIT_E;
   #X71a := (#S71a OR (#X71a AND NOT #S72a AND NOT #S73a)) AND NOT #FORCE_INIT_E;
   #X72a := (#S72a OR (#X72a AND NOT #S73a)) AND NOT #FORCE_INIT_E;
   #X73a := (#S73a OR (#X73a AND NOT #S70a)) AND NOT #FORCE_INIT_E;

   #STOP_ACT := #X71a;
   #FORCE_INIT := #FORCE_INIT_E OR #X72a;
   #FORCE_CURRENT := #FORCE_CURRENT_E OR #X71a;
   #RESET_ALARMA := #X73a;
   #T1(IN:=#X72,
       PT:=T#1s
   );
   #T2(IN := #X73,
       PT := T#1s
   );
   #T3(IN := #X76,
       PT := T#3s
   );


   // PRODUCCIÓN
   #S70 := ("FirstScan" OR (#X76 AND #T3.Q)) AND NOT #FORCE_CURRENT;
   #S71 := (#X70 AND #Act_Proceso) AND NOT #FORCE_CURRENT;
   #S72 := (#X71 AND #S5) AND NOT #FORCE_CURRENT;
   #S73 := (#X72 AND #T1.Q) AND NOT #FORCE_CURRENT;
   #S74 := (#X73 AND #T2.Q) AND NOT #FORCE_CURRENT;
   #S75 := (#X74 AND #Pieza_Empaquetada) AND NOT #FORCE_CURRENT;
   #S76 := (#X75 AND #SigMaqLibre) AND NOT #FORCE_CURRENT;


   #X70 := (#S70 OR #X70 AND (NOT #S71)) OR #FORCE_INIT;
   #X71 := (#S71 OR #X71 AND (NOT #S72)) AND NOT #FORCE_INIT;
   #X72 := (#S72 OR #X72 AND (NOT #S73)) AND NOT #FORCE_INIT;
   #X73 := (#S73 OR #X73 AND (NOT #S74)) AND NOT #FORCE_INIT;
   #X74 := (#S74 OR #X74 AND (NOT #S75)) AND NOT #FORCE_INIT;
   #X75 := (#S75 OR #X75 AND (NOT #S76)) AND NOT #FORCE_INIT;
   #X76 := (#S76 OR #X76 AND (NOT #S70)) AND NOT #FORCE_INIT;



   #Maq_Libre := #X70 AND NOT #STOP_ACT;
   #QC5 := (#X71 OR #X72 OR #Mantenimiento_Cinta OR #vaciado_cinta) AND NOT #STOP_ACT;
   #QC6 := (#X71 OR #X72 OR #Mantenimiento_Cinta OR #vaciado_cinta) AND NOT #STOP_ACT;
   #QC7 := (#X71 OR #X72 OR #X73 OR #X76 OR #Mantenimiento_Cinta OR #vaciado_cinta) AND NOT #STOP_ACT;
   #QCLAMP := (#X73 OR #X74 OR #Mantenimiento_Clamper) AND NOT #STOP_ACT;
   #QCLAMP_SUB := (#X76 OR #Mantenimiento_SubirClamp OR #vaciado_subclamp) AND NOT #STOP_ACT;
   #Act_SIG_MAQ := #X76 AND NOT #STOP_ACT;
   #HayPieza := #X74 AND NOT #STOP_ACT;
   //#Pieza_Empaquetada := X62 AND NOT STOP_ACT;

   #T1a(IN:=#X71,
        PT:=T#20s);


   //#Alarma_1 := (#Alarma_1 OR (#T1a.Q)) AND NOT #RESET_ALARMA;
   //#Alarma_2 := (#Alarma_2 OR (#X33 AND #T2.Q)) AND NOT RESET_ALARMA;

   //#Alarma := (#Alarma_1) AND NOT (#FORCE_INIT OR #RESET_ALARMA);
   //#Alarma_Maquina := #Alarma;
END_FUNCTION_BLOCK

FUNCTION_BLOCK "Grafcet_10_Final_1"   // FB31, SCL
{ S7_Optimized_Access := 'TRUE' }
VERSION : 0.1
   VAR_INPUT
      Act_Maquina : Bool;
      S_Pres : Bool;
      S1 : Bool;
      Sig_Maq_Libre : Bool;
      Mantenimiento_Cintas : Bool;
      vaciado_cinta : Bool;
      Pieza_Rec : Bool;
      Reset : Bool;
      Resume : Bool;
      CI : Bool;
      Emergencia : Bool;
   END_VAR
   VAR_OUTPUT
      Emisor : Bool;
      Emisor_2 : Bool;
      Maq_Libre : Bool;
      QC1A : Bool;
      QC1B : Bool;
      Act_SIG_MAQ : Bool;
      Alarma_Maquina : Bool;
   END_VAR
   VAR_IN_OUT
      Alarma_1 : Bool;
      Alarma_2 : Bool;
   END_VAR
   VAR
      S10 : Bool;
      S11 : Bool;
      S12 : Bool;
      S13 : Bool;
      S14 : Bool;
      S15 : Bool;
      X10 : Bool;
      X15 : Bool;
      X11 : Bool;
      X12 : Bool;
      X13 : Bool;
      X14 : Bool;
      S10e : Bool;
      S11e : Bool;
      S12e : Bool;
      X10e : Bool;
      X11e : Bool;
      X12e : Bool;
      FORCE_INIT : Bool;
      FORCE_INIT_E : Bool;
      FORCE_CURRENT_E : Bool;
      S10a : Bool;
      S11a : Bool;
      S12a : Bool;
      S13a : Bool;
      X10a : Bool;
      X11a : Bool;
      X12a : Bool;
      X13a : Bool;
      FORCE_CURRENT : Bool;
      STOP_ACT : Bool;
      RESET_ALARMA : Bool;
      Alarma : Bool;
      S11b : Bool;
      X11b : Bool;
      T1a : TON_TIME;
      trig_PR : R_TRIG;
   END_VAR
BEGIN
   //Flancos


   // EMERGENCIA
   #S10e := (#X12e AND #CI) OR "FirstScan";
   #S11e := #X10e AND "Emergencia";
   #S12e := #X11e;

   #X10e := #S10e OR (#X10e AND NOT #S11e);
   #X11e := #S11e OR (#X11e AND NOT #S12e);
   #X12e := #S12e OR (#X12e AND NOT #S10e);

   #FORCE_INIT_E := #X11e;
   #FORCE_CURRENT_E := #X12e;


   // ALARMAS
   #S10a := (#X13a AND NOT #FORCE_CURRENT_E) OR "FirstScan";
   #S11a := (#X10a AND #Alarma) AND NOT #FORCE_CURRENT_E;
   #S12a := (#X11a AND #Reset) AND NOT #FORCE_CURRENT_E;
   #S13a := (#X12a OR (#X11a AND #Resume)) AND NOT #FORCE_CURRENT_E;

   #X10a := #S10a OR (#X10a AND NOT #S11a) OR #FORCE_INIT_E;
   #X11a := (#S11a OR (#X11a AND NOT #S12a AND NOT #S13a)) AND NOT #FORCE_INIT_E;
   #X12a := (#S12a OR (#X12a AND NOT #S13a)) AND NOT #FORCE_INIT_E;
   #X13a := (#S13a OR (#X13a AND NOT #S10a)) AND NOT #FORCE_INIT_E;

   #STOP_ACT := #X11a;
   #FORCE_INIT := #FORCE_INIT_E OR #X12a;
   #FORCE_CURRENT := #FORCE_CURRENT_E OR #X11a;
   #RESET_ALARMA := #X13a;

   #trig_PR(CLK:=#Pieza_Rec);

   // PRODUCCIÓN
   #S10 := ("FirstScan" OR (#X15 AND #trig_PR.Q)) AND NOT #FORCE_CURRENT;
   #S11 := (#X10 AND #Act_Maquina) AND NOT #FORCE_CURRENT;
   #S11b := (#X11 AND (#S_Pres )) AND NOT #FORCE_CURRENT;
   #S12 := (#X11b AND( NOT #S_Pres )) AND NOT #FORCE_CURRENT;
   #S13 := (#X12 AND #S1) AND NOT #FORCE_CURRENT;
   #S14 := (#X13 AND #Sig_Maq_Libre) AND NOT #FORCE_CURRENT;
   #S15 := (#X14 AND NOT #S1) AND NOT #FORCE_CURRENT;


   #X10 := (#S10 OR #X10 AND (NOT #S11)) OR #FORCE_INIT;
   #X11 := (#S11 OR #X11 AND (NOT #S11b)) AND NOT #FORCE_INIT;
   #X11b := (#S11b OR #X11b AND (NOT #S12)) AND NOT #FORCE_INIT;
   #X12 := (#S12 OR #X12 AND (NOT #S13 AND NOT #S14)) AND NOT #FORCE_INIT;
   #X13 := (#S13 OR #X13 AND (NOT #S14)) AND NOT #FORCE_INIT;
   #X14 := (#S14 OR #X14 AND (NOT #S15)) AND NOT #FORCE_INIT;
   #X15 := (#S15 OR #X15 AND (NOT #S10)) AND NOT #FORCE_INIT;


   #Maq_Libre := #X10 AND NOT #STOP_ACT;
   #Emisor_2 := ("Proceso_Activo") AND NOT #STOP_ACT;
   #Emisor := ("Proceso_Activo") AND NOT #STOP_ACT;
   //#Emisor_2 := (#X11 AND NOT #S_Pres) AND NOT #STOP_ACT;
   //#Emisor := (#X11 AND NOT #S_Pres) AND NOT #STOP_ACT;
   #QC1A := (#X11 OR #X11b OR #Mantenimiento_Cintas OR #vaciado_cinta)  AND NOT #STOP_ACT;
   #QC1B := ( #X11b OR #X12 OR #X14 OR #Mantenimiento_Cintas OR #vaciado_cinta) AND NOT #STOP_ACT;
   #Act_SIG_MAQ := #X14 AND NOT #STOP_ACT;


   #T1a(IN:=#X14,
        PT:=T#5s);
   //#Alarma_1 := #Alarma_1 OR (#X12 AND #S_Pres)AND NOT #RESET_ALARMA;
   //#Alarma_2 := #Alarma_2 OR (#T1a.Q) AND NOT #RESET_ALARMA;
   //#Alarma := (#Alarma_1 OR #Alarma_2) AND NOT (#FORCE_INIT OR #RESET_ALARMA);
   //#Alarma_Maquina := #Alarma;
END_FUNCTION_BLOCK

FUNCTION_BLOCK "Grafcet_20_2_FInal"   // FB32, SCL
{ S7_Optimized_Access := 'TRUE' }
VERSION : 0.1
   VAR_INPUT
      Act_Proceso : Bool;
      SigMaqLibre : Bool;
      SA_Bueno : Bool;
      SA_Malo : Bool;
      SB : Bool;
      Mantenimiento_Cintas : Bool;
      Mantenimiento_Transfers : Bool;
      vaciado_cinta : Bool;
      vaciado_trans : Bool;
      CI : Bool;
      Reset : Bool;
      Resume : Bool;
   END_VAR
   VAR_OUTPUT
      Maq_Libre : Bool;
      QC2 : Bool;
      QTRANS : Bool;
      Act_SIG_MAQ_Buena : Bool;
      Act_SIG_MAQ_Mala : Bool;
      Pieza_Rec : Bool;
   END_VAR
   VAR
      S20 : Bool;
      S21 : Bool;
      S22 : Bool;
      S23 : Bool;
      S24 : Bool;
      S22b : Bool;
      S23b : Bool;
      X20 : Bool;
      X21 : Bool;
      X22 : Bool;
      X22b : Bool;
      X23 : Bool;
      X23b : Bool;
      X24 : Bool;
      S20a : Bool;
      S21a : Bool;
      S22a : Bool;
      S23a : Bool;
      X20a : Bool;
      X21a : Bool;
      X22a : Bool;
      X23a : Bool;
      S20e : Bool;
      S21e : Bool;
      S22e : Bool;
      X20e : Bool;
      X21e : Bool;
      X22e : Bool;
      FORCE_INIT : Bool;
      FORCE_INIT_E : Bool;
      FORCE_CURRENT : Bool;
      FORCE_CURRENT_E : Bool;
      STOP_ACT : Bool;
      RESET_ALARMA : Bool;
      Alarma : Bool;
      T1 : TON_TIME;
   END_VAR
BEGIN


   // EMERGENCIA
   #S20e := (#X22e AND #CI) OR "FirstScan";
   #S21e := #X20e AND "Emergencia";
   #S22e := #X21e;

   #X20e := #S20e OR (#X20e AND NOT #S21e);
   #X21e := #S21e OR (#X21e AND NOT #S22e);
   #X22e := #S22e OR (#X22e AND NOT #S20e);

   #FORCE_INIT_E := #X21e;
   #FORCE_CURRENT_E := #X22e;


   // ALARMAS
   #S20a := (#X23a AND NOT #FORCE_CURRENT_E) OR "FirstScan";
   #S21a := (#X20a AND #Alarma) AND NOT #FORCE_CURRENT_E;
   #S22a := (#X21a AND #Reset) AND NOT #FORCE_CURRENT_E;
   #S23a := (#X22a OR (#X21a AND #Resume)) AND NOT #FORCE_CURRENT_E;

   #X20a := #S20a OR (#X20a AND NOT #S21a) OR #FORCE_INIT_E;
   #X21a := (#S21a OR (#X21a AND NOT #S22a AND NOT #S23a)) AND NOT #FORCE_INIT_E;
   #X22a := (#S22a OR (#X22a AND NOT #S23a)) AND NOT #FORCE_INIT_E;
   #X23a := (#S23a OR (#X23a AND NOT #S20a)) AND NOT #FORCE_INIT_E;

   #STOP_ACT := #X21a;
   #FORCE_INIT := #FORCE_INIT_E OR #X22a;
   #FORCE_CURRENT := #FORCE_CURRENT_E OR #X21a;
   #RESET_ALARMA := #X23a;
   #T1(IN:=#X24,
       PT:=T#2s);




   // PRODUCCIÓN
   #S20 := ("FirstScan" OR (#X22b AND NOT #SA_Bueno AND NOT #SA_Malo AND NOT #SB) OR (#X23b AND NOT #SA_Malo AND NOT #SA_Bueno AND NOT #SB) OR (#X24 AND #T1.Q) ) AND NOT #FORCE_CURRENT;
   #S21 := (#X20 AND #Act_Proceso) AND NOT #FORCE_CURRENT;
   #S22 := (#X21 AND #SA_Bueno AND #SA_Malo AND #SB) AND NOT #FORCE_CURRENT;
   #S22b := (#X22 AND #SigMaqLibre) AND NOT #FORCE_CURRENT;
   #S23 := (#X21 AND #SA_Malo AND NOT #SA_Bueno AND #SB) AND NOT #FORCE_CURRENT;
   #S23b := (#X23 AND #SigMaqLibre) AND NOT #FORCE_CURRENT;
   #S24 := (#X21 AND #SB AND #SA_Bueno AND NOT #SA_Malo) AND NOT #FORCE_CURRENT;



   #X20 := (#S20 OR #X20 AND (NOT #S21)) OR #FORCE_INIT;
   #X21 := (#S21 OR #X21 AND (NOT #S22 AND NOT #S23 AND NOT #S24)) AND NOT #FORCE_INIT;
   #X22 := (#S22 OR #X22 AND (NOT #S22b)) AND NOT #FORCE_INIT;
   #X22b := (#S22b OR #X22b AND (NOT #S20)) AND NOT #FORCE_INIT;
   #X23 := (#S23 OR #X23 AND (NOT #S23b)) AND NOT #FORCE_INIT;
   #X23b := (#S23b OR #X23b AND (NOT #S20)) AND NOT #FORCE_INIT;
   #X24 := (#S24 OR #X24 AND (NOT #S20)) AND NOT #FORCE_INIT;



   #Maq_Libre := #X20 AND NOT #STOP_ACT;
   #QC2 := (#X21 OR #X22b OR #X23b OR #Mantenimiento_Cintas OR #vaciado_cinta) AND NOT #STOP_ACT;
   #QTRANS := (#X24 OR #Mantenimiento_Transfers OR #vaciado_trans)AND NOT #STOP_ACT;
   #Act_SIG_MAQ_Buena := #X22b AND NOT #STOP_ACT;
   #Act_SIG_MAQ_Mala := #X23b AND NOT #STOP_ACT;
   #Pieza_Rec := (#X22 OR #X23 OR #X24) AND NOT #STOP_ACT;
END_FUNCTION_BLOCK

ORGANIZATION_BLOCK "Main"   // OB1, LAD, ProgramCycle
TITLE = "Main Program Sweep (Cycle)"
{ S7_Optimized_Access := 'TRUE' }
VERSION : 0.1
   VAR_INPUT
      Initial_Call : Bool;   // Initial call of this OB
      Remanence : Bool;   // =True, if remanent data are available
   END_VAR
   VAR_TEMP   // added for the SCL form of the ladder/FBD networks
      _w1 : Bool;
      _w2 : Bool;
      _w3 : Bool;
      _w4 : Bool;
      _w5 : Bool;
      _w6 : Bool;
      _w7 : Bool;
   END_VAR
BEGIN

REGION Network 1: Grafctet Principal
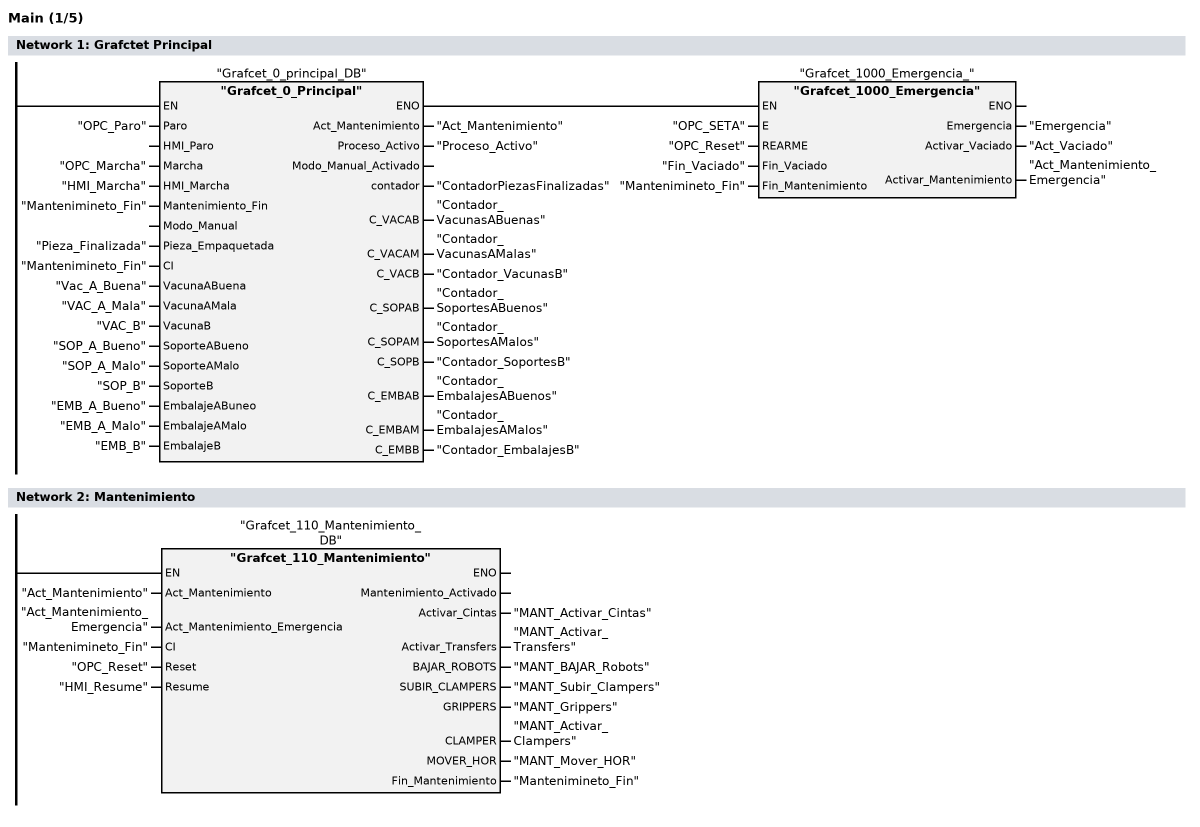
   RUNG wire#powerrail
      "Grafcet_0_principal_DB"(Paro := "OPC_Paro", HMI_Paro :=, Marcha := "OPC_Marcha", HMI_Marcha := "HMI_Marcha", Mantenimiento_Fin := "Mantenimineto_Fin", Modo_Manual :=, Pieza_Empaquetada := "Pieza_Finalizada", CI := "Mantenimineto_Fin", VacunaABuena := "Vac_A_Buena", VacunaAMala := "VAC_A_Mala", VacunaB := "VAC_B", SoporteABueno := "SOP_A_Bueno", SoporteAMalo := "SOP_A_Malo", SoporteB := "SOP_B", EmbalajeABuneo := "EMB_A_Bueno", EmbalajeAMalo := "EMB_A_Malo", EmbalajeB := "EMB_B", Act_Mantenimiento => "Act_Mantenimiento", Proceso_Activo => "Proceso_Activo", Modo_Manual_Activado =>, contador => "ContadorPiezasFinalizadas", C_VACAB => "Contador_VacunasABuenas", C_VACAM => "Contador_VacunasAMalas", C_VACB => "Contador_VacunasB", C_SOPAB => "Contador_SoportesABuenos", C_SOPAM => "Contador_SoportesAMalos", C_SOPB => "Contador_SoportesB", C_EMBAB => "Contador_EmbalajesABuenos", C_EMBAM => "Contador_EmbalajesAMalos", C_EMBB => "Contador_EmbalajesB")
      "Grafcet_1000_Emergencia_"("E" := "OPC_SETA", REARME := "OPC_Reset", Fin_Vaciado := "Fin_Vaciado", Fin_Mantenimiento := "Mantenimineto_Fin", Emergencia => "Emergencia", Activar_Vaciado => "Act_Vaciado", Activar_Mantenimiento => "Act_Mantenimiento_Emergencia")
   END_RUNG
   // the same network as SCL:
   "Grafcet_0_principal_DB"(Paro := "OPC_Paro",   // "Grafcet_0_Principal"
                           Marcha := "OPC_Marcha",
                           HMI_Marcha := "HMI_Marcha",
                           Mantenimiento_Fin := "Mantenimineto_Fin",
                           Pieza_Empaquetada := "Pieza_Finalizada",
                           CI := "Mantenimineto_Fin",
                           VacunaABuena := "Vac_A_Buena",
                           VacunaAMala := "VAC_A_Mala",
                           VacunaB := "VAC_B",
                           SoporteABueno := "SOP_A_Bueno",
                           SoporteAMalo := "SOP_A_Malo",
                           SoporteB := "SOP_B",
                           EmbalajeABuneo := "EMB_A_Bueno",
                           EmbalajeAMalo := "EMB_A_Malo",
                           EmbalajeB := "EMB_B",
                           Act_Mantenimiento => "Act_Mantenimiento",
                           Proceso_Activo => "Proceso_Activo",
                           contador => "ContadorPiezasFinalizadas",
                           C_VACAB => "Contador_VacunasABuenas",
                           C_VACAM => "Contador_VacunasAMalas",
                           C_VACB => "Contador_VacunasB",
                           C_SOPAB => "Contador_SoportesABuenos",
                           C_SOPAM => "Contador_SoportesAMalos",
                           C_SOPB => "Contador_SoportesB",
                           C_EMBAB => "Contador_EmbalajesABuenos",
                           C_EMBAM => "Contador_EmbalajesAMalos",
                           C_EMBB => "Contador_EmbalajesB",
                           ENO => #_w1);
   IF #_w1 THEN
       "Grafcet_1000_Emergencia_"("E" := "OPC_SETA",   // "Grafcet_1000_Emergencia"
                               REARME := "OPC_Reset",
                               Fin_Vaciado := "Fin_Vaciado",
                               Fin_Mantenimiento := "Mantenimineto_Fin",
                               Emergencia => "Emergencia",
                               Activar_Vaciado => "Act_Vaciado",
                               Activar_Mantenimiento => "Act_Mantenimiento_Emergencia");
   END_IF;
END_REGION

REGION Network 2: Mantenimiento
   RUNG wire#powerrail
      "Grafcet_110_Mantenimiento_DB"(Act_Mantenimiento := "Act_Mantenimiento", Act_Mantenimiento_Emergencia := "Act_Mantenimiento_Emergencia", CI := "Mantenimineto_Fin", Reset := "OPC_Reset", Resume := "HMI_Resume", Mantenimiento_Activado =>, Activar_Cintas => "MANT_Activar_Cintas", Activar_Transfers => "MANT_Activar_Transfers", BAJAR_ROBOTS => "MANT_BAJAR_Robots", SUBIR_CLAMPERS => "MANT_Subir_Clampers", GRIPPERS => "MANT_Grippers", CLAMPER => "MANT_Activar_Clampers", MOVER_HOR => "MANT_Mover_HOR", Fin_Mantenimiento => "Mantenimineto_Fin")
   END_RUNG
   // the same network as SCL:
   "Grafcet_110_Mantenimiento_DB"(Act_Mantenimiento := "Act_Mantenimiento",   // "Grafcet_110_Mantenimiento"
                           Act_Mantenimiento_Emergencia := "Act_Mantenimiento_Emergencia",
                           CI := "Mantenimineto_Fin",
                           Reset := "OPC_Reset",
                           Resume := "HMI_Resume",
                           Activar_Cintas => "MANT_Activar_Cintas",
                           Activar_Transfers => "MANT_Activar_Transfers",
                           BAJAR_ROBOTS => "MANT_BAJAR_Robots",
                           SUBIR_CLAMPERS => "MANT_Subir_Clampers",
                           GRIPPERS => "MANT_Grippers",
                           CLAMPER => "MANT_Activar_Clampers",
                           MOVER_HOR => "MANT_Mover_HOR",
                           Fin_Mantenimiento => "Mantenimineto_Fin");
END_REGION

